// TwinCAT 3 PLC project CrimperProject
// ProgramVersion: 3.1.4023.0
// CompilerDefines: VISU_USEWSTRING, CRIMP_IO_TEST
// libraries:
//   CmpBitmapPool, * (System)
//   Tc2_Standard, * (Beckhoff Automation GmbH)
//   Tc2_System, * (Beckhoff Automation GmbH)
//   Tc2_Utilities, * (Beckhoff Automation GmbH)
//   Tc3_Module, * (Beckhoff Automation GmbH)
//   VisuDialogs, * (System)
//   VisuSymbols,3.5.10.0,System
// project tree:
//   DUTs/ DUT_Errors.TcDUT, DUT_Device.TcDUT, DUT_RunTime.TcDUT
//   / GlobalTextList.TcGTLO, ImagePool.TcIPO (not stored), PlcTask.TcTTO, VISU_TASK.TcTTO
//   GVLs/ CVL.TcGVL, DB6.TcGVL, GVL.TcGVL, IO.TcGVL, RVL.TcGVL, VAT.TcGVL
//   POUs/Helper/ FB_CalcXY.TcPOU, FB_INPUT_HANDLER.TcPOU, FB_MY_BLINK.TcPOU, P_GetTime.TcPOU, TSV.TcPOU
//   POUs/HMI/ P_HmiHandling.TcPOU
//   POUs/Initialization/ P_InitOnce.TcPOU
//   POUs/Language/ P_RestoreCurrentLanguage.TcPOU, P_SaveCurrentLanguage.TcPOU
//   POUs/ MAIN.TcPOU
//   POUs/MainPous/F20_Ablauf/AusstossVerzoegerung/ P_DecAusStossV.TcPOU, P_IncAusstossV.TcPOU
//   POUs/MainPous/F20_Ablauf/DrahtHalterDruck/ P_DecDruck.TcPOU, P_IncDruck.TcPOU
//   POUs/MainPous/F20_Ablauf/ F_AblaufketteLeerfahren.TcPOU, FB_AblaufketteNormal.TcPOU, P_AblaufReset.TcPOU, FB_AllesInSollposition.TcPOU, F_Endstellung.TcPOU, F_Ventile.TcPOU, P_Ablauf.TcPOU
//   POUs/MainPous/F20_Ablauf/SollwertRuettelTopf/ P_DecSollRuettel.TcPOU, P_IncSollRuettel.TcPOU
//   POUs/MainPous/FC24_Sortierer/ F_Leerfahren.TcPOU, F_Sortierer.TcPOU, F_Vereinzelung.TcPOU, P_Sortierer.TcPOU
//   POUs/MainPous/FC2_Betriebsarten/ P_BlinktaktTastleuchten.TcPOU, F_EndschalterBruecken.TcPOU, P_FlankenErzeugen.TcPOU, F_StartStopTipp.TcPOU, P_Betriebsarten.TcPOU, P_InputHandling.TcPOU, P_OutputHandling.TcPOU
//   POUs/MainPous/FC3_FehlerAllg/ F_Aufstarten.TcPOU, F_AusloeseschalterDauermeldung.TcPOU, F_Doppelmeldung.TcPOU, F_FehlerAufgetreten.TcPOU, F_GetErrorsAsDWORD.TcPOU, FB_KontrolleEndschalter.TcPOU, F_KontrollZeiten.TcPOU, F_ResetEndSchalterFehler.TcPOU, F_ResetErrors.TcPOU, F_StoerungsbitsAuswerten.TcPOU, P_FehlerAllgemein.TcPOU
//   POUs/MainPous/FC4_TpKommunikation/ F_AnzeigeNiedriegePrio.TcPOU, F_AnzeigeSollpositionsFehler.TcPOU, F_AuswertungBefehlstastenVonTP.TcPOU, F_SAFETY_AnzeigenHohePrio.TcPOU, F_SAFETY_AnzeigenHohePrio_Neu.TcPOU, F_SignaldauerVonTastleuchte_MaschEinAuswerten.TcPOU, P_OnResetClick.TcPOU, P_TpKommunikation.TcPOU
//   POUs/MainPous/FC95_StatusAnzeige/ P_StatusAnzeige.TcPOU
//   POUs/MainPous/FC99_LetzterFC/ P_LetzterFC.TcPOU
//   VISUs/ Ausstossverz.TcVIS, BetrAnzeigeListe.TcTLO, DrahthalterDruck.TcVIS, IO_Visu01.TcVIS, IO_Visu02.TcVIS, Menu.TcVIS, Probelauf.TcVIS, Rezeptur.TcVIS, Sprache.TcVIS, OutTest.TcVIS, SensorBruecken.TcVIS, Start.TcVIS, Stueckzahl.TcVIS, Total.TcVIS, VisualizationManager.TcVMO (not stored)
// real-time tasks:
//   TASK PlcTask: cycle T#20ms, priority 20, ADS port 350
//   TASK VISU_TASK: cycle T#200000us, priority 30, ADS port 351
//   TASK Standard: cycle T#1ms, priority 1, ADS port 352
//   TASK ELM-Task: cycle T#1ms, priority 2, ADS port 353
// I/O:
//   DEVICE Gerät 3 (EtherCAT), AmsNetId 172.18.216.102.4.1
//     Klemme 1 (EK1100-0008) [EK1100-0008 EtherCAT-Koppler M8 (2A E-Bus)]
//       Klemme 2 (EL1809) [EL1809 16K. Dig. Eingang 24V, 3ms]
//       Klemme 3 (EL2809) [EL2809 16K. Dig. Ausgang 24V, 0.5A]
//       Klemme 4 (EL4122) [EL4122 2K. Ana. Ausgang 4-20mA, 16bit]
//       Klemme 5 (EL2911) [EL2911,  Potential supply terminal (10 A) with 4 Ch. Safety Inputs, TwinSAFE]
//         modules: Module 2 (FSOUT), Module 3 (DEVICEIO), Module 4 (FSLOGIC)
//       Klemme 7 (ELM3702-0000) [ELM3702-0000 2K. Ana. Eingang +/-60V, +/-20mA, TC, RTD, Messbrückenauswertung (DMS), IEPE, 24 bit, hochgenau]
//       Klemme 6 (EL9011) [EL9011 Endklemme]
// variable links:
//   CrimperProject/CrimperProject Instance <-> Device 3 (EtherCAT)/Term 1 (EK1100-0008)/Term 2 (EL1809)
//     PlcTask Inputs/IO.inAbisoliererIstLINKS <-> Channel 8/Input
//     PlcTask Inputs/IO.inAbisoliererIstRUECK <-> Channel 7/Input
//     PlcTask Inputs/IO.inAbisoliererIstVORN <-> Channel 6/Input
//     PlcTask Inputs/IO.inAbisoliererIstZU <-> Channel 5/Input
//     PlcTask Inputs/IO.inAusloeseSchalter <-> Channel 4/Input
//     PlcTask Inputs/IO.inAusstossenVORN <-> Channel 14/Input
//     PlcTask Inputs/IO.inCrimpEinheitIstRUECK <-> Channel 13/Input
//     PlcTask Inputs/IO.inCrimpEinheitIstVORN <-> Channel 12/Input
//     PlcTask Inputs/IO.inCrimpZangeIstOFFEN <-> Channel 10/Input
//     PlcTask Inputs/IO.inCrimpZangeIstZU <-> Channel 9/Input
//     PlcTask Inputs/IO.inDrahthalterIstOffen <-> Channel 3/Input
//     PlcTask Inputs/IO.inKontaktIstGefallen <-> Channel 11/Input
//     PlcTask Inputs/IO.inKontaktSchiebenVORN <-> Channel 15/Input
//     PlcTask Inputs/IO.inMagazinGEFUELLT <-> Channel 16/Input
//     PlcTask Inputs/IO.inResetNotHalt <-> Channel 1/Input
//     PlcTask Inputs/IO.inStart <-> Channel 2/Input
//     PlcTask Inputs/IO.inWord0 @bit {1..15} <-> Channel {2..16}/Input  (15 links)
//     PlcTask Inputs/IO.inWord0 <-> Channel 1/Input
//   CrimperProject/CrimperProject Instance <-> Device 3 (EtherCAT)/Term 1 (EK1100-0008)/Term 3 (EL2809)
//     PlcTask Outputs/IO.outMldTasteStart <-> Channel 2/Output
//     PlcTask Outputs/IO.outNotHaltReset <-> Channel 1/Output
//     PlcTask Outputs/IO.outResA1_2 <-> Channel 3/Output
//     PlcTask Outputs/IO.outY10DrahthaltFuehrungZU <-> Channel 16/Output
//     PlcTask Outputs/IO.outY11SortierLuft <-> Channel 6/Output
//     PlcTask Outputs/IO.outY1Ausstossen <-> Channel 7/Output
//     PlcTask Outputs/IO.outY2KontaktVereinzelung <-> Channel 8/Output
//     PlcTask Outputs/IO.outY3KontaktSchieben <-> Channel 9/Output
//     PlcTask Outputs/IO.outY4CrimpEinheitVOR <-> Channel 10/Output
//     PlcTask Outputs/IO.outY5AbisolierNachLINKS <-> Channel 11/Output
//     PlcTask Outputs/IO.outY6AbisoliererZU <-> Channel 12/Output
//     PlcTask Outputs/IO.outY7AbfallRUNTER <-> Channel 13/Output
//     PlcTask Outputs/IO.outY8AbisoliererRUECK <-> Channel 14/Output
//     PlcTask Outputs/IO.outY9CrimperZU <-> Channel 15/Output
//   CrimperProject/CrimperProject Instance <-> Device 3 (EtherCAT)/Term 1 (EK1100-0008)/Term 4 (EL4122)
//     PlcTask Outputs/IO.outSollwertDruckVentil <-> Channel 2/Output
//     PlcTask Outputs/IO.outSollwertRuettelTopf <-> Channel 1/Output
//   CrimperProject/CrimperProject Instance <-> Device 3 (EtherCAT)/Term 1 (EK1100-0008)/Term 5 (EL2911)
//     PlcTask Inputs/IO.safeOutHauptLuft <-> StandardInputs/Standard Out Var 6
//     PlcTask Inputs/IO.safeOutNotHalt <-> StandardInputs/Standard Out Var 11
//     PlcTask Inputs/IO.safeOutSchutzTueren <-> StandardInputs/Standard Out Var 12
//     PlcTask Outputs/IO.safetyRUN <-> StandardOutputs/Standard In Var 2

CONFIGURATION CrimperProject
    RESOURCE PLC ON TwinCAT3
        TASK PlcTask(INTERVAL := T#20ms, PRIORITY := 20);
        TASK VISU_TASK(INTERVAL := T#200000us, PRIORITY := 30);
        PROGRAM MAIN WITH PlcTask : MAIN;
        PROGRAM VisuElems_Visu_Prg WITH VISU_TASK : VisuElems.Visu_Prg;
    END_RESOURCE
END_CONFIGURATION

// ---- DUTs/DUT_Errors.TcDUT
TYPE DUT_Errors :
STRUCT

    //M104.0
	DrahthltNichtOffen : BIT; //(ehem. M104.0) Drahthalter nicht offen, BetrAnzeigeListe.ID 600
	DrahthltNichtZu : BIT; //(ehem. M104.1) Drahthalter nicht zu, BetrAnzeigeListe.ID 601
	AusloesSchaltDauerMldg: BIT;//(ehem. M104.2) -- Auslöseschalter Dauermelung, BetrAnzeigeListe.ID 602
	AbisolierNichtOffen : BIT; //(ehem. M104.3) Abisolierer nicht offen, BetrAnzeigeListe.ID 603
	AbisolierNichtZu : BIT; //(ehem. M104.4) Abisolierer nicht zu, BetrAnzeigeListe.ID 604
	DoppelMlgAbisoVornRueck : BIT; //(ehem. M104.5) Doppelmeldung Abisolierer vorn+rück, BetrAnzeigeListe.ID 605
	AbisolierNichtVorn : BIT; //(ehem. M104.6) Abisolierer nicht vorn, BetrAnzeigeListe.ID 606
	AbisolierNichtRueck : BIT; //(ehem. M104.7) Abisolierer nicht rück (abisoliert), BetrAnzeigeListe.ID 607
	
	//M105.0
	AbisolierNichtLinks : BIT; //(ehem. M105.0) Abisolierer nicht links (aus Arbeitsraum) , BetrAnzeigeListe.ID 608
	AbisolierNichtRechts : BIT; //(ehem. M105.1) Abisolierer nicht rechts, BetrAnzeigeListe.ID 609
	DoppelMlgCrimpzZuOffen : BIT; //(ehem. M105.2) Doppelmeldung Crimpzange zu+offen, BetrAnzeigeListe.ID 610
	CrimpZangeNichtZu : BIT; //(ehem. M105.3) Crimpzange nicht zu, BetrAnzeigeListe.ID 611
	CrimpZangeNichtOffen : BIT; //(ehem. M105.4) Crimpzange nicht offen, BetrAnzeigeListe.ID 612
	KontaktNichtGefallen : BIT; //(ehem. M105.5) !! nur xls File !!, BetrAnzeigeListe.ID 613
	DauerMlgKontaktGefallen : BIT; //(ehem. 105.6) !! nur xls File !!, BetrAnzeigeListe.ID 614
	DoppelMlgCrimpEinhVornZurueck : BIT; //(ehem. M105.7) Doppelmeldung Crimpeinheit vorn+rück, BetrAnzeigeListe.ID 615
	
	//M106.0
	CrimpeinheitNichtVorn : BIT; //(ehem. M106.0)Crimpeinheit nicht vorn, BetrAnzeigeListe.ID 616
	CrimpeinheitNichtRueck : BIT; //(ehem. M106.1) Crimpeinheit nicht rück, BetrAnzeigeListe.ID 617
	KontaktSchiebenNichtVorn : BIT; //(ehem. M106.2) Kontakt-Schieben nicht vorn, BetrAnzeigeListe.ID 618
	KontaktSchiebenNichtRueck : BIT; //(ehem. M106.3) Kontakt-Schieben nicht rück, BetrAnzeigeListe.ID 619
	AusstossenNichtVorn : BIT; //(ehem. M106.4) Ausstoßen nicht vorn, BetrAnzeigeListe.ID 620
	AusstossenNichtRueck : BIT; //(ehem. M106.5) Ausstoßen nicht rück, BetrAnzeigeListe.ID 621
	r106_6 : BIT; //Reserve, war in AWL nicht belegt, BetrAnzeigeListe.ID 622
	WartungsZaehlErreicht : BIT; //(ehem. M106.7) Wartungs-Zähler, hat Vorwahl eicht, BetrAnzeigeListe.ID 623
	
	//M107.0
	StueckZaehlErreicht : BIT; //(ehem. M107.0 Stückzahl-Vorwahl eicht), BetrAnzeigeListe.ID 624
	r107_1 : BIT; //Reserve, war in AWL nicht belegt, BetrAnzeigeListe.ID 625 
	r107_2 : BIT; //Reserve, war in AWL nicht belegt, BetrAnzeigeListe.ID 626
	r107_3 : BIT; //Reserve, war in AWL nicht belegt, BetrAnzeigeListe.ID 627
	r107_4 : BIT; //Reserve, war in AWL nicht belegt, BetrAnzeigeListe.ID 628
	r107_5 : BIT; //Reserve, war in AWL nicht belegt, BetrAnzeigeListe.ID 629
	r107_6 : BIT; //Reserve, war in AWL nicht belegt, BetrAnzeigeListe.ID 630
	r107_7 : BIT; //Reserve, war in AWL nicht belegt, BetrAnzeigeListe.ID 631   

END_STRUCT
END_TYPE

// ---- DUTs/DUT_Device.TcDUT
TYPE DUT_Device :
STRUCT
	wID:WORD; (* Geräte ID *)
		
	rIN_LO:REAL; (* REAL in Wert unten *)
	rIN_HI:REAL; (* REAL in Wert oben *)
	nOUT_LO:UINT; (* RAW out Wert unten *)
	nOUT_HI:UINT; (* RAW out Wert oben *)
	
	dFakt_A:REAL; (* Faktor 'a' in Y=aX + b *)
	dSmd_B:REAL; (* Summand 'b' in Y=aX + b *)
	
	sDevName:STRING(50); (* Gerätename *)

END_STRUCT
END_TYPE

// ---- DUTs/DUT_RunTime.TcDUT
TYPE DUT_RunTime :
STRUCT
	seconds:INT;
	mins:INT;
	hours:DINT;
END_STRUCT
END_TYPE

// ---- GVLs/CVL.TcGVL
{attribute 'qualified_only'}
VAR_GLOBAL CONSTANT

(* LogLevels: 0-Nothing, 1-ErrOnly, 2-Warnings, 4-Info , 8-All *)
ERROR:WORD:=1;
WARNING:WORD:=2;
INFO:WORD:=4;
TRACE:WORD:=8;
	
enableIN1_2 : BOOL := TRUE; // (ehem. M11.0, insecDrahthalterIstOffen)

BTN_STOP : INT := 130; // Stop-Taste im Start-Menü ??? original ??? noch klären

BTRART_RESET : INT := 800; // Bertriebsarten-Reset 
RESET_BUTTON : INT := 801; // Reset-Button
MAGAZIN_LEER : INT := 810; // Magazin Leerfahren
SORTIER_LEER : INT := 820; // Sortierer Leerfahren
CRIMP_EINRICHTEN : INT := 830; //Crimpen Einrichten
NUR_ABISOLIER : INT := 840; // Nur Abisolieren
PROBE_OHNE_KONT : INT := 850; // Probelauf ohne Kontakt
PROBE_OHNE_CRIMP : INT := 860; // Probelauf ohne Crimpen
PROBE_OHNE_LITZE : INT :=870; // Probelauf ohne Litze
END_VAR

// ---- GVLs/DB6.TcGVL
{attribute 'qualified_only'}
VAR_GLOBAL RETAIN
	
	rAusstossverz : REAL := 0.0; //ehem. in DB6.w134
	nAusstossverz : INT := 0; //NEU-NBT

	diStueck_Vorwahl: DINT := 10000;//ehem. in DB6.d64Stueck_Vorwahl
	diStueck_Fertig: DINT := 0; //ehem. in DB6.d68Stueck_Fertig
	diStueck_Noch: DINT := 10000;
	iStueck_pro_Minute: INT := 0;
	
	diStueck_Total : DINT := 0;
	
	
	diTotalZaehler: DINT := 0; // ehem. in DB6.d140
	diTagesZaehler: DINT := 0; // ehem. in DB6.d144
	
	diWartZaehlVorwahl: DINT := 0; // Vorwahl Wartung, ehem. in DB6.d148
	diWartungsZaehler: DINT := 0; // ehem. in DB6.d152
	
	diReinigung_Vorw: DINT := 10000; //ehem. in DB6.d80
	diReinigung_Zaehl: DINT := 0; //ehem. in DB6.d84
	
	rDrahthalterSchliessdruck : REAL := 0.5; //Umwandlung in F_Ventile() - wDrahthalterSchliessdruck := REAL_TO_WORD(DINT_TO_REAL(DB6.d376) * 2.730000E+003);
	
	
	iSortierer : INT := 50; // Sortierer-Sollwert (Analog), war w132_Sortierer
	
	w226_Betr_Anz_Wert : INT := 0; // Betriebs-Anzeige-Wert Bedeutung noch unklar!!!
	w230 : INT := 0; // Signaldauer-Wert von PNOZ Bedeutung noch unklar!!!
	w228_Bef_Tast_Wert : INT := 0;
	
	outWordAlt : WORD; //ehem. in DB6.d408 -- Zuw.v. AW0
	
	d0 : DWORD := 0;
	
	runTime : DUT_RunTime;  //ehem. in DB6.d160 ff., todo versteckt. Reset?
	
	
	//Test später raus --- Begin ---
	
	frceY11SortierLuft 			: BOOL; //EL1809-A1.5
	frceY1Ausstossen 			: BOOL;
	frceY2KontaktVereinzelung 	: BOOL; //EL1809-A1.7
	frceY3KontaktSchieben	 	: BOOL; //EL1809-A1.8
	frceY4CrimpEinheitVOR	 	: BOOL; //EL1809-A1.9
	frceY5AbisolierNachLINKS	: BOOL; //EL1809-A1.10
	frceY6AbisoliererZU		 	: BOOL; //EL1809-A1.11
	frceY7AbfallRUNTER		 	: BOOL; //EL1809-A1.12
	frceY8AbisoliererRUECK	 	: BOOL; //EL1809-A1.13
	frceY9CrimperZU			 	: BOOL; //EL1809-A1.14
	frceY10DrahthaltFuehrungZU	: BOOL; //EL1809-A1.15
	
	//Test später raus --- End ---
END_VAR

// ---- GVLs/GVL.TcGVL
{attribute 'qualified_only'}
VAR_GLOBAL
	firstCycle : BOOL;	
	
	insecResetNotHalt			: BOOL; //result of P_InputHandling.E1_0
	insecTasterStart 			: BOOL; //result of P_InputHandling.E1_1
	insecDrahthalterIstOffen 	: BOOL; //result of P_InputHandling.E1_2
	insecAusloeseSchalter		: BOOL; //result of P_InputHandling.E1_3
	insecAbisoliererIstZU		: BOOL; //result of P_InputHandling.E1_4
	insecAbisoliererIstVORN		: BOOL; //result of P_InputHandling.E1_5
	insecAbisoliererIstRUECK	: BOOL; //result of P_InputHandling.E1_6
	insecAbisoliererIstLINKS	: BOOL; //result of P_InputHandling.E1_7
	
	insecCrimpZangeIstZU		: BOOL; //result of P_InputHandling.E1_8
	insecCrimpZangeIstOFFEN		: BOOL; //result of P_InputHandling.E1_9
	insecKontaktIstGefallen		: BOOL; //result of P_InputHandling.E1_10
	insecCrimpEinheitIstVORN	: BOOL; //result of P_InputHandling.E1_11
	insecCrimpEinheitIstRUECK	: BOOL; //result of P_InputHandling.E1_12
	insecAusstossenVORN			: BOOL; //result of P_InputHandling.E1_13
	insecKontaktSchiebenVORN	: BOOL; //result of P_InputHandling.E1_14
	insecMagazinGEFUELLT		: BOOL; //result of P_InputHandling.E1_15
	
	
	inTmpResetNotHalt			: BOOL; //result of P_InputHandling.E1_0
	inTmpTasterStart 			: BOOL; //result of P_InputHandling.E1_1
	inTmpDrahthalterIstOffen 	: BOOL; //result of P_InputHandling.E1_2
	inTmpAusloeseSchalter		: BOOL; //result of P_InputHandling.E1_3
	inTmpAbisoliererIstZU		: BOOL; //result of P_InputHandling.E1_4
	inTmpAbisoliererIstVORN		: BOOL; //result of P_InputHandling.E1_5
	inTmpAbisoliererIstRUECK	: BOOL; //result of P_InputHandling.E1_6
	inTmpAbisoliererIstLINKS	: BOOL; //result of P_InputHandling.E1_7
	
	inTmpCrimpZangeIstZU		: BOOL; //result of P_InputHandling.E1_8
	inTmpCrimpZangeIstOFFEN		: BOOL; //result of P_InputHandling.E1_9
	inTmpKontaktIstGefallen		: BOOL; //result of P_InputHandling.E1_10
	inTmpCrimpEinheitIstVORN	: BOOL; //result of P_InputHandling.E1_11
	inTmpCrimpEinheitIstRUECK	: BOOL; //result of P_InputHandling.E1_12
	inTmpAusstossenVORN			: BOOL; //result of P_InputHandling.E1_13
	inTmpKontaktSchiebenVORN	: BOOL; //result of P_InputHandling.E1_14
	inTmpMagazinGEFUELLT		: BOOL; //result of P_InputHandling.E1_15
	
	
	
	tof00Test : TOF;
	(* ehem. T0 ersetzt durch BLINK *)
	tonTasteStartOnErr : TON;	// (ehem. T1 SE->TON) Verzögerung Taste Start
	//T2 Verz.v. Taste Stop, existierte im AWL-Text nicht
	tonFehlerKontrMaschine  : TON; // (ehem. T3) Fehler-Kontr.Maschine (keine Bewegung)
	
	tonTasteStart : TON; // (ehem. T11) Taster-Start Verz. in F_Aufstarten(), für StörMldgLöschen
	tonBetrAnzeigReset : TON; // (ehem. T14) Verz. Betriebs-Anzeigen-Reset
	tonEndschalterBrueck : TON; // (ehem. T15) Verz. Endschalter-Brückung
	tonAusloesDauermld : TON; // (ehem. T16) Kontr.Auslöseschalter Dauermeldung
	tsvVereinzelZeit : TSV; // (ehem. T17) AWL-SV: Vereinzelungs-Zeit, Zeit mit verlängertem Impuls
	tonKontaktIstGefallen : TON; // (ehem. T18) Verz.v. E1.10 Kontakt gefallen
	tsvKontauswurf : TSV;	// (ehem. T19) AWL-SV: Kontaktauswurf nach Einschalten, Zeit mit verlängertem Impuls
	
	tofAblVerzProbelauf : TOF; 	// (ehem. T20) Ablauf-Verz.bei Probelauf
	ton2terVersuch : TON; //(ehem. T21) Verz. 2ter Vereinzelungs-Versuch
	tonAusstoss : TON; // (ehem. T22) Ausstoß-Verzögerung
	tonKontaktIstZuLangeEin : TON; //NEU Fehlererzeugung für DauermeldungKontaktGefallen
	
	tofCrimpzangeOffen : TOF; // (ehem. T31) Verl. E1.9 Crimpzange offen
	tofMagazGefuellt : TOF; // (ehem. T32) Verl. E1.15 Magazin gefüllt
	tofMagazGefuellt2 : TON; // (ehem. T33) 2te Verl. T32 E1.15 Magazin gefüllt
	
	tofBetrStdZaehl : TOF; // (ehem. T34)  Verl. 5 Minuten für Betriebstunden-Zähler, Zeit mit Ausschaltverzögerung
	tofMagazLeerFahr : TOF; // // (ehem. T41) Takt für Magazin leerfahren, wird 2x verwendet???

	
	tonResetNotHalt : TON; // Neu: check rote Stop-Taste
	//tonPnozEntprell  : TON; //(ehem. T70) PNOZ ???Entprell??
	//tofPnozSigLen : TOF; // (ehem. T71) PNOZ Signaldauer ???
	tonSAFETYok : TON; // (ehem. T72) Verzögerung Alles Ok von PNOZ, tonOkPNOZ
	
	
	tonDrahthaltOffen : TON; // (ehem. T110) Brücke EL1809-E1.2 Drahthalter offen
	tonAbisoliererIstZU : TON; // (ehem. T112) Brücke EL1809-E1.4 Abisolierer zu
	tonAbisoliererIstVORN : TON; // (ehem. T113) Brücke EL1809-E1.5 Abisolierer vorn
	tonAbisoliererIstRUECK : TON; // (ehem. T114) Brücke EL1809-E1.6 Abisolierer rück (abisoliert)
	tonAbisoliererIstLINKS : TON; // (ehem. T115) Brücke EL1809-E1.7 Abisolierer links (aus Arbeitsraum)
	tonCrimpZangeIstZU : TON; // (ehem. T116) Brücke EL1809-E1.8 Crimpzange zu
	tonCrimpZangeIstOFFEN : TON; // (ehem. T117) Brücke EL1809-E1.9 Crimpzange offen
	
	tonBrKontaktIstGefallen : TON; // (ehem. T120) Brücke EL1809-E1.10 Kontakt gefallen
	tonCrimpEinheitIstVORN : TON; // (ehem. T121) Brücke EL1809-E1.11 Crimpeinheit vorn
	tonKontaktSchiebenVORN : TON; // (ehem. T122) Brücke EL1809-E1.14 Kontakt-Schieben vorn
	tonAusstossenVORN : TON; // (ehem. T123) Brücke EL1809-E1.13 Ausstoßen vorn
	tonCrimpEinheitIstRUECK : TON; // (ehem. T124) Brücke EL1809-E1.12 Crimpeinheit rück
	
	bTEMP : BOOL;
	
	MW0 : WORD; //Bedeutung noch Unklar
	
	
	
	//MD20 : DWORD; //Bedeutung noch Unklar
	MD80 : DWORD; // +Fs ED0, wird offensichtlich nicht verwendet!	
		
	
	//MD100 : DWORD; //Bedeutung noch Unklar, irgendwas mit Störungen
	//MD104 : DWORD; //Bedeutung noch Unklar, irgendwas mit Störungen
	//MD108 : DWORD; //Bedeutung noch Unklar, irgendwas mit Störungen
	//MD112 : DWORD; //Bedeutung noch Unklar, irgendwas mit Störungen
	//MD116 : DWORD; //Bedeutung noch Unklar, irgendwas mit Störungen
	//MD120 : DWORD; //Bedeutung noch Unklar, irgendwas mit Störungen
	
	BetrAnzeigeIdx : INT; // (ehem. MW14 : WORD) // enthält Betriebs-Anzeige-Bits (jetzt Index)
	BetrAnzeigeTmp : INT;
	TopfWert : UINT;
	
	SolPosErrorIdx : WORD;
	EinzelschrittIdx : WORD;
	
	devSortierer : DUT_Device;
	devDruckVentil : DUT_Device;
	calcDev : FB_CalcXY;
	
	errs : DUT_Errors;
	errsAsDword : DWORD;
	zeigeFehler : BOOL;
	
END_VAR

// ---- GVLs/IO.TcGVL
{attribute 'qualified_only'}
VAR_GLOBAL

	//EL1809 16xDE (-10K1)
	inResetNotHalt				AT%I* : BOOL; //EL1809-E1.0 - roteTaste, LowAktiv
	inStart 					AT%I* : BOOL; //EL1809-E1.1 (ehem. E0.0)
	inDrahthalterIstOffen 		AT%I* : BOOL; //EL1809-E1.2 (ehem. E1.0)
	inAusloeseSchalter			AT%I* : BOOL; //EL1809-E1.3 (ehem. E1.1), wenn Draht in Aufnahme
	inAbisoliererIstZU			AT%I* : BOOL; //EL1809-E1.4 (ehem. E1.2)
	inAbisoliererIstVORN		AT%I* : BOOL; //EL1809-E1.5 (ehem. E1.3)
	inAbisoliererIstRUECK		AT%I* : BOOL; //EL1809-E1.6 (ehem. E1.4)
	inAbisoliererIstLINKS		AT%I* : BOOL; //EL1809-E1.7 (ehem. E1.5)
	
	inCrimpZangeIstZU			AT%I* : BOOL; //EL1809-E1.8 (ehem. E1.6)
	inCrimpZangeIstOFFEN		AT%I* : BOOL; //EL1809-E1.9 (ehem. E1.7)
	inKontaktIstGefallen		AT%I* : BOOL; //EL1809-E1.10 (ehem. E2.0)
	inCrimpEinheitIstVORN		AT%I* : BOOL; //EL1809-E1.11 (ehem. E2.1)
	inCrimpEinheitIstRUECK		AT%I* : BOOL; //EL1809-E1.12 (ehem. E2.4)
	inAusstossenVORN			AT%I* : BOOL; //EL1809-E1.13 (ehem. E2.3)
	inKontaktSchiebenVORN		AT%I* : BOOL; //EL1809-E1.14 (ehem. E2.2)
	inMagazinGEFUELLT			AT%I* : BOOL; //EL1809-E1.15 (ehem. E2.5)
	
	inWord0 					AT%I* : WORD; //Eingangswort komplett für EL1809-E1.
	
	
	
	//EL1809 16xDA (-10K4)
	outNotHaltReset 			AT%Q* : BOOL; //EL2809-A1.0
	//ToDo umben. 'TastleuchteStart'	
	outMldTasteStart			AT%Q* : BOOL; //EL2809-A1.1 (ehem. A0.0),Meldeleuchte Taste Start
	outResA1_2					AT%Q* : BOOL; //EL2809-A1.2
	//resA1.3
	//resA1.4
	outY11SortierLuft 			AT%Q* : BOOL; //EL2809-A1.5  (ehem. A0.1), toDo umben. BlasLuftSortierer...
	outY1Ausstossen 			AT%Q* : BOOL; //EL2809-A1.6  (ehem. A0.6)
	outY2KontaktVereinzelung	AT%Q* : BOOL; //EL2809-A1.7  (ehem. A0.7)
	outY3KontaktSchieben	 	AT%Q* : BOOL; //EL2809-A1.8  (ehem. A1.0)
	outY4CrimpEinheitVOR	 	AT%Q* : BOOL; //EL2809-A1.9  (ehem. A1.1)
	outY5AbisolierNachLINKS	 	AT%Q* : BOOL; //EL2809-A1.10 (ehem. A1.2)
	outY6AbisoliererZU		 	AT%Q* : BOOL; //EL2809-A1.11 (ehem. A1.3)
	outY7AbfallRUNTER		 	AT%Q* : BOOL; //EL2809-A1.12 (ehem. A1.4)
	outY8AbisoliererRUECK	 	AT%Q* : BOOL; //EL2809-A1.13 (ehem. A1.5)
	outY9CrimperZU			 	AT%Q* : BOOL; //EL2809-A1.14 (ehem. A1.6)
	outY10DrahthaltFuehrungZU	AT%Q* : BOOL; //EL2809-A1.15 (ehem. A1.7)
	
	
	//EL4122 (-10K6)
	outSollwertRuettelTopf		AT%Q* : UINT; //EL4122-AAW1
	//ToDo umbenennen bis in Klemme 4 outDrahthaltSchliessdrSoll
	outSollwertDruckVentil		AT%Q* : UINT; //EL4122-AAW2 Drahthalter Schliessdruck Sollwert
	
	//EL2911 (-10K6.1)
	safeInModuleFault			AT%I* : BOOL; //EL2911 In-Module-Fault
	safeOutNotHalt				AT%I* : BOOL; //EL2911 geklonter Ausgang des Not-Halt-AND Objekts
	safeOutSchutzTueren			AT%I* : BOOL; //EL2911 geklonter Ausgang des SchutzTueren-AND Objekts

	
	safeOutModuleFault			AT%I* : BOOL; //EL2911 Out-Module-Fault
	safeOutHauptLuft			AT%I* : BOOL; //EL2911-OUT1
	
	safetyErrAcknowledge 		AT%Q* : BOOL; //
	safetyRUN 					AT%Q* : BOOL; //EL2911 verlinkt mit dem Safety-Projekt 
	
	
	outWord0 : WORD; //Ausgangswort komplett für EL2809-E1. (selbst gefüllt)
END_VAR

// ---- GVLs/RVL.TcGVL
{attribute 'qualified_only'}
VAR_GLOBAL PERSISTENT
	
	e10Online : BOOL := TRUE; //ON-, OFF-line switch E1.0
	e11Online : BOOL := TRUE;
	e12Online : BOOL := TRUE;
	e13Online : BOOL := TRUE;
	e14Online : BOOL := TRUE;
	e15Online : BOOL := TRUE;
	e16Online : BOOL := TRUE;
	e17Online : BOOL := TRUE;
	
	e18Online : BOOL := TRUE;
	e19Online : BOOL := TRUE;
	e110Online : BOOL := TRUE; //ON-, OFF-line switch E1.10
	e111Online : BOOL := TRUE;
	e112Online : BOOL := TRUE;
	e113Online : BOOL := TRUE;
	e114Online : BOOL := TRUE;
	e115Online : BOOL := TRUE;
	
	e10OffMode : BOOL := FALSE; //Low-, High-switch for Offline mode E1.0
	e11OffMode : BOOL := FALSE;
	e12OffMode : BOOL := FALSE;
	e13OffMode : BOOL := FALSE;
	e14OffMode : BOOL := FALSE;
	e15OffMode : BOOL := FALSE;
	e16OffMode : BOOL := FALSE;
	e17OffMode : BOOL := FALSE;
		
	e18OffMode : BOOL := FALSE;
	e19OffMode : BOOL := FALSE;
	e110OffMode : BOOL := FALSE; //Low-, High-switch for Offline mode E1.10
	e111OffMode : BOOL := FALSE;
	e112OffMode : BOOL := FALSE;
	e113OffMode : BOOL := FALSE;
	e114OffMode : BOOL := FALSE;
	e115OffMode : BOOL := FALSE;

	
	currLogLevel : WORD := 0;
	currLanguage : STRING(10);
	
	
	//sBr: Sensor Brücke TRUE = eingeschalet, Sensor überbrückt
	sBrDrahthalterIstOffen 		: BOOL; //Brücke für: EL1809-E1.2
	sBrAusloeseSchalter			: BOOL; //Brücke für: EL1809-E1.3
	sBrAbisoliererIstZU			: BOOL; //Brücke für: EL1809-E1.4
	sBrAbisoliererIstVORN		: BOOL; //Brücke für: EL1809-E1.5
	sBrAbisoliererIstRUECK		: BOOL; //Brücke für: EL1809-E1.6
	sBrAbisoliererIstLINKS		: BOOL; //Brücke für: EL1809-E1.7
	
	sBrCrimpZangeIstZU			: BOOL; //Brücke für: EL1809-E1.8
	sBrCrimpZangeIstOFFEN		: BOOL; //Brücke für: EL1809-E1.9
	sBrKontaktIstGefallen		: BOOL; //Brücke für: EL1809-E1.10
	sBrCrimpEinheitIstVORN		: BOOL; //Brücke für: EL1809-E1.11
	sBrCrimpEinheitIstRUECK		: BOOL; //Brücke für: EL1809-E1.12
	sBrAusstossenVORN			: BOOL; //Brücke für: EL1809-E1.13
	sBrKontaktSchiebenVORN		: BOOL; //Brücke für: EL1809-E1.14
	sBrMagazinGEFUELLT			: BOOL; //Brücke für: EL1809-E1.15
END_VAR

// ---- GVLs/VAT.TcGVL
{attribute 'qualified_only'}
VAR_GLOBAL

	//MB5 : BYTE; // +F Blinktakt-Generator
	//MB6 : BYTE; // kein Gebrauch, nur 0-Initialisierung
	b00Test : BOOL := FALSE;
	//M0 : BYTE;
	(*
	0.0 -- frei
	0.1 -- frei
	0.2 -- 2te Ablauf-Freigabe
	0.3 -- Tipp, Einzel-Schritt
	0.4 -- frei 
	0.5 -- Bedingung für Ablauf-Freigabe
	0.6 -- SR Start
	0.7 -- Sammel-Störung
	*)
	bZweitAblaufFreig : BOOL; //ehem. M0.2 -- 2te Ablauf-Freigabe
 	bEinzelSchritt : BOOL;	//ehem. M0.3 -- Tipp, Einzel-Schritt
	bAblaufFreigabe : BOOL; //ehem. M0.5 -- Bedingung für Ablauf-Freigabe
	bSrStart : BOOL; 		//ehem. M0.6 -- SR Start
	bSammelStoerung : BOOL;	//ehem. M0.7 -- Sammel-Störung

	//M1 : BYTE;
	//1.0 -- frei 
	//1.1 -- frei
	//1.2 -- frei
	//1.3 -- RS Stop
	bRsStop : BOOL; //ehem. M1.3 -- RS Stop
	
	//M3 : BYTE;
	//3.0 -- Alles in Sollposition
	//3.1 -- PNOZ old
	//3.2 -- frei 
	//3.3 -- frei
	//3.4 -- frei
	//3.5 -- frei
	//3.6 -- frei
	//3.7 -- frei
	bAllesInSollPos : BOOL; //(ehem. M3.0 -- Alles in Sollposition)
	bResetNotHalt_Old : BOOL; //(ehem. M3.1 -- PNOZ old)
	
	//M4 : BYTE; //Blinktakt-Generator
	//4.0 -- 8-Hz Blinktakt
	//4.1 -- 4-Hz Blinktakt
	//4.2 -- 2-Hz Blinktakt
	//4.3 -- 1-Hz Blinktakt
	//4.4 -- 0.5-Hz Blinktakt (alle 2 sec)
	//4.5 -- 0.25-Hz Blinktakt (alle 4 sec)
	//4.6 -- 0.125-Hz Blinktakt (alle 8 sec)
	//4.7 -- frei
	
	byBlinkTakt : BYTE := 0; //Blinktakt-Generator (ehem. M4)
	//4.0 -- 8-Hz Blinktakt
	//4.1 -- 4-Hz Blinktakt
	//4.2 -- 2-Hz Blinktakt
	//4.3 -- 1-Hz Blinktakt
	//4.4 -- 0.5-Hz Blinktakt (alle 2 sec)
	//4.5 -- 0.25-Hz Blinktakt (alle 4 sec)
	//4.6 -- 0.125-Hz Blinktakt (alle 8 sec)
	//4.7 -- frei
		
	//M5 : BYTE;
	//5.0 
	//5.1
	//5.2
	//5.3 -- +F 1-Hz Blinktakt
	//5.4
	//5.5
	//5.6
	//5.7
	
	b1HzFlanke : BOOL; //(ehem. M5.3 -- +F 1-Hz Blinktakt)
	
	//M6 : BYTE;
	//6.0 -- +F Reset-Button
	bFlkResetButton : BOOL := FALSE; //(ehem. M6.0 -- +F Reset-Button)
	
	
	//M8 : BYTE; //MB8
	//8.0	M8.0 NormalCrimp
	//8.1	Magazin Leerfahren
	//8.2	Sortierer Leerfahren
	//8.3	"M8.3 CrimpEinr
	//8.4	"M8.4 NurAbisolieren
	//8.5	Probelauf ohne Kontakt
	//8.6	"M8.6 ohneCrmpen
	//8.7	"M8.7 Probelauf ohne Litze
	
	bNormalCrimp : BOOL; 			//(ehem. M8.0 NormalCrimp)
	bMagazinLeerfahren : BOOL; 		//(ehem. M8.1 Magazin Leerfahren)
	bSortiererLeerfahren : BOOL;	//(ehem. M8.2 Sortierer Leerfahren)
	bCrimpEinrichten : BOOL; 		//(ehem. M8.3 Crimp Einrichten)
	bNurAbisolieren : BOOL; 		//(ehem. M8.4 Nur Abisolieren)
	bProbelOhneKontakt : BOOL;		//(ehem. M8.5 Probelauf ohne Kontakt)
	bProbelOhneCrimpen : BOOL; 		//(ehem. M8.6 ohne Crimpen)
	bProbelOhneLitze : BOOL; 		//(ehem. M8.7 Probelauf ohne Litze)
	
	//M9 : BYTE;
	//9.0 -- mit Sortier-Blasen
	//9.1
	//9.2
	//9.3 
	//9.4
	//9.5
	//9.6
	//9.7
	bSortiererBlasen : BOOL; //(ehem. M9.0 -- mit Sortier-Blasen)
	bSortiererBlasenAlt : BOOL;
	sortierTextID : INT := 1000;
	
	//M11 : BYTE; --- RVL.sBrDrahthalterIstOffen...
	//11.0 -- Brücke E1.0 Drahthalter offen
	//11.1 -- Brücke E1.1 Auslöseschalter
	//11.2 -- Brücke E1.2 Abisolierer zu
	//11.3 -- Brücke E1.3 Abisolierer vorn
	//11.4 -- Brücke E1.4 Abisolierer rück (abisoliert)
	//11.5 -- Brücke E1.5 Abisolierer links (aus Arbeitsraum)
	//11.6 -- Brücke E1.6 Crimpzange zu
	//11.7 -- Brücke E1.7 Crimpzange offen
	
	// M12 : BYTE; --- RVL.sBrKontaktIstGefallen...
	//12.0 -- Brücke E2.0 Kontakt gefallen
	//12.1 -- Brücke E2.1 Crimpeinheit vorn
	//12.2 -- Brücke E2.2 Kontakt-Schieben vorn
	//12.3 -- Brücke E2.3 Ausstoßen vorn
	//12.4 -- Brücke E2.4 Crimpeinheit rück
	//12.5 -- Brücke E2.5 Magazin gefüllt
	//12.6
	//12.7
	
	//M14 : BYTE;
	//14.0 -- A55 Kontakt nicht gefallen
	//14.1
	//14.2
	//14.3
	//14.4
	//14.5
	//14.6
	//14.7
	bA55KontaktNichtGefallen:BOOL; //(ehem. M14.0 A55 Kontakt nicht gefallen)
	
	//M20 : BYTE; //Schrittkette
	//20.0 -- Drahthalter + Drahtführung zu
	//20.1 -- Abisolierer zu
	//20.2 -- Abisolierer rück
	//20.3 -- Abisolierer nach links + Abisolierer auf
	//20.4 -- Crimpeinheit vor
	//20.5 -- Crimpeinheit zu
	//20.6 -- Drahthalter + Drahtführung auf
	//20.7 -- Crimpzange auf + Abisoliereinheit vor
	
	bDrahtHalterUndFuehrungZU : BOOL; //(ehem. M20.0 -- Drahthalter + Drahtführung zu)
	bAbisoliererZU : BOOL; //(ehem. M20.1 -- Abisolierer zu )
	bAbisoliererRUECK : BOOL; //(ehem. M20.2 -- Abisolierer rück )
	bAbisoliererLINKSundAUF : BOOL; //(ehem. M20.3 -- Abisolierer nach links + Abisolierer auf )
	bCrimpeinheitVOR : BOOL; //(ehem. M20.4 --Crimpeinheit vor)
	bCrimpenZU : BOOL; //(ehem. M20.5 --Crimpeinheit zu)
	bDrahtHalterUndFuehrungAUF : BOOL; //(ehem. M20.6 --Drahthalter + Drahtführung auf)
	bCrZangeAUF_AisolierVOR : BOOL; //(ehem. M20.7 -- Crimpzange auf + Abisoliereinheit vor)
	
	
	//M21 : BYTE;
	//21.0  -- Ausstoßen vor
	//21.1 -- Crimpeinheit rück
	//21.2 -- Abisolierer nach rechts + Kontakt-Schieben rück
	//21.3
	//21.4
	//21.5
	//21.6 -- Aktueller Ablauf ohne Crimpen
	//21.7 -- Kontakt-Anforderung
	bAusstossenVOR : BOOL; //(ehem. M21.0 Ausstoßen vor)
	bCrimpeinheitRUECK : BOOL; //(ehem. M21.1 Ausstoßen vor)
	bAbisoNachRE_KontSchiebRUECK : BOOL; //(ehem. M21.2 Abisolierer nach rechts + Kontakt-Schieben rück)
	
	
	bAktAblaufOhneCr : BOOL;	//(ehem. M21.6  -- Aktueller Ablauf ohne Crimpen)
	bKontaktAnforderung : BOOL; //(ehem. M21.7  -- Kontakt-Anforderung)
	
	//M22 : BYTE;
	//22.0 -- Abisolierer nach Links Leerf-o-Crimpen
	//22.1 -- Crimpeinheit vor Leerf-o-Crimpen
	//22.2 -- Vereinzelung takten od.Crimpen
	//22.3 -- Crimpeinheit rück Leerf-o-Crimpen
	//22.4 -- frei
	//22.5 -- frei
	//22.6 -- Crimpen beim Einstellen
	//22.7 -- Endstellung
	bAbisoliererNachLinksLoC : BOOL; //(ehem. M22.0 Abisolierer nach Links Leerfahren-ohne-Crimpen)
	bCrimpEinheitVorLoC : BOOL; //(ehem. M22.1 Crimpeinheit vor Leerfahren-ohne-Crimpen)
	bVereinzelungTakten  : BOOL; //(ehem. M22.2 takten od.Crimpen)
	bCrimpEinheitRueckLoC : BOOL; //(ehem. M22.3 rück Leerfahren-ohne-Crimpen)
	//frei
	bCrimpenZuBeiEinstellen : BOOL; //(ehem. M22.6 Crimpen zu bei Einstellen Leerfahren-ohne-Crimpen)
	bEndstellung : BOOL; //(ehem. M22.7 Endstellung)
	
	//M23 : BYTE;
	//23.0 -- Takt für Vereinzelung bei Leerfahren
	//23.1 -- Zylinder sollen IN Leerfahrstellung
	//23.2 -- Zylinder sollen AUS Leerfahrstellung
	//23.3 -- S&R 2ter Vereinzelungs-Versuch
	//23.4
	//23.5
	//23.6
	//23.7
	bTaktVereinzLeerF : BOOL; //(ehem. M23.0 Takt für Vereinzelung bei Leerfahren)
	bZylINLeerFahrt : BOOL; //(ehem. M23.1 Zylinder sollen IN Leerfahrstellung)
	bZylAUSLeerFahrt : BOOL; //(ehem. M23.2 Zylinder sollen AUS Leerfahrstellung)
	bSr2terVereinzVersuch : BOOL; //(ehem. M23.3 S&R 2ter Vereinzelungs-Versuch)
	
	//M24 : BYTE;
	//24.0 
	//24.1 -- Zuw.v.T21 2ter Vereinzelungs-Versuch
	//24.2 -- +F 2ter Vereinzelungs-Versuch
	//24.3
	//24.4
	//24.5
	//24.6
	//24.7
	bFlk2terVersuch : BOOL; //(ehem. M24.2) +F 2ter Vereinzelungs-Versuch
	
	//M60 : BYTE; //MB60
	
	//M80 : BYTE;
	//80.0 //+F E0.0 Taste Start
	bFlkTasteStart : BOOL; //(ehem. M80.0) +F E0.0 Taste Start
	bFlkTasteStop : BOOL; //NEU
	
	//M81 : BYTE;
	//81.0 
	//81.1 -- +F E1.1 Auslöseschalter
	//81.2
	//81.3
	//81.4
	//81.5
	//81.6
	//81.7
	bFlankeAusloeseschalter : BOOL;  //(ehem. M81.1) +F E1.1 Auslöseschalter
	
	//M82 : BYTE;
	//82.0 
	//82.1 
	//82.2
	//82.3
	//82.4
	//82.5 -- +F E2.5 Magazin gefüllt
	//82.6
	//82.7
	bFlankeMagazGefuellt : BOOL; //(ehem. M82.5) +F E2.5 Magazin gefüllt
	
	(*
	
	//M104 : BYTE;
	//104.0 -- Drahthalter nicht offen
	//104.1 -- Drahthalter nicht zu
	//104.2 -- Auslöseschalter Dauermelung
	//104.3 -- Abisolierer nicht offen
	//104.4 -- Abisolierer nicht zu
	//104.5 -- Doppelmeldung Abisolierer vorn+rück
	//104.6 -- Abisolierer nicht vorn
	//104.7 -- Abisolierer nicht rück (abisoliert)
	errDrahthltNichtOffen : BOOL; //(ehem. M104.0) Drahthalter nicht offen
	errDrahthltNichtZu : BOOL; //(ehem. M104.1) Drahthalter nicht zu
	errAusloesSchaltDauerMldg: BOOL;//(ehem. M104.2) -- Auslöseschalter Dauermelung
	errAbisolierNichtOffen : BOOL; //(ehem. M104.3) Abisolierer nicht offen
	errAbisolierNichtZu : BOOL; //(ehem. M104.4) Abisolierer nicht zu
	errDoppelMlgAbisoVornRueck : BOOL; //(ehem. M104.5) Doppelmeldung Abisolierer vorn+rück
	errAbisolierNichtVorn : BOOL; //(ehem. M104.6) Abisolierer nicht vorn
	errAbisolierNichtRueck : BOOL; //(ehem. M104.7) Abisolierer nicht rück (abisoliert)
		
	
	//M105 : BYTE;
	//105.0 -- Abisolierer nicht links (aus Arbeitsraum)
	//105.1 -- Abisolierer nicht rechts
	//105.2 -- Doppelmeldung Crimpzange zu+offen
	//105.3 -- Crimpzange nicht zu
	//105.4 -- Crimpzange nicht offen
	//105.5 -- Kontakt nicht gefallen 
	//105.6
	//105.7 -- Doppelmeldung Crimpeinheit vorn+rück
	errAbisolierNichtLinks : BOOL; //(ehem. M105.0) Abisolierer nicht links (aus Arbeitsraum)
	errAbisolierNichtRechts : BOOL; //(ehem. M105.1) Abisolierer nicht rechts
	errDoppelMlgCrimpzZuOffen : BOOL; //(ehem. M105.2) Doppelmeldung Crimpzange zu+offen
	errCrimpZangeNichtZu : BOOL; //(ehem. M105.3) Crimpzange nicht zu
	errCrimpZangeNichtOffen : BOOL; //(ehem. M105.4) Crimpzange nicht offen
	errKontaktNichtGefallen : BOOL; //(ehem. M105.5) !! nur xls File !! --
	errDauermeldungKontaktGefallen : BOOL; //(ehem. 105.6) !! nur xls File !! --
	errDoppelMlgCrimpEinhVornZurueck : BOOL; //(ehem. M105.7) Doppelmeldung Crimpeinheit vorn+rück
	
	
	//M106 : BYTE;
	//106.0 -- Crimpeinheit nicht vorn
	//106.1 -- Crimpeinheit nicht rück
	//106.2 -- Kontakt-Schieben nicht vorn
	//106.3 -- Kontakt-Schieben nicht rück
	//106.4 -- Ausstoßen nicht vorn
	//106.5 -- Ausstoßen nicht rück
	//106.6
	//106.7 -- Wartungs-Zähler, hat Vorwahl erreicht, weiter mit Reset
	errCrimpeinheitNichtVorn : BOOL; //(ehem. M106.0)Crimpeinheit nicht vorn
	errCrimpeinheitNichtRueck : BOOL; //(ehem. M106.1) Crimpeinheit nicht rück
	errKontaktSchiebenNichtVorn : BOOL; //(ehem. M106.2) Kontakt-Schieben nicht vorn
	errKontaktSchiebenNichtRueck : BOOL; //(ehem. M106.3) Kontakt-Schieben nicht rück
	errAusstossenNichtVorn : BOOL; //(ehem. M106.4) Ausstoßen nicht vorn
	errAusstossenNichtRueck : BOOL; //(ehem. M106.5) Ausstoßen nicht rück
	//106.6
	bWartungsZaehlErreicht : BOOL := FALSE; //(ehem. M106.7) Wartungs-Zähler, hat Vorwahl erreicht
	
	//M107 : BYTE;
	//107.0 -- Stückzahl-Vorwahl erreicht
	//107.1 -- 
	//107.2 -- 
	//107.3 -- 
	//107.4 -- 
	//107.5
	//107.6
	//107.7
	bStueckZaehlErreicht : BOOL := FALSE; //(ehem. M107.0 Stückzahl-Vorwahl erreicht)
	*)
	aw4Sortierer : WORD;
END_VAR

// ---- POUs/MAIN.TcPOU
PROGRAM MAIN
VAR
	//rTrig : R_TRIG;
	dwTmp : DWORD;
END_VAR

P_InitOnce(); // NBT-NEU 

P_GetTime(); // NBT-NEU 

P_RestoreCurrentLanguage(); // NBT-NEU 

P_InputHandling(); // NBT-NEU 

P_TpKommunikation(); //ehem. FC4 -- OK

P_Betriebsarten(); //ehem. FC2 -- OK

P_Ablauf(); //ehem. FC20 -- OK -- 500er ID-Bereich

P_Sortierer(); //ehem. FC24 -- OK

P_FehlerAllgemein(); //ehem. FC3 -- OK -- 600er ID-Bereich

P_StatusAnzeige(); //ehem. FC95

//P_LetzterFC(); //ehem. FC99

P_OutputHandling(); // OK

P_HmiHandling(); //NBT-NEU

METHOD M_Log : DINT
VAR_INPUT
	reqLevel : WORD; (* 0-Nothing, 1-ErrOnly, 2-Warnings, 4-Info , 8-Verbose *)
	objectName : STRING(40);
	sMsg	: T_MaxString;(* Message string *)
	errNo : UDINT := 16#FFFFFFFF;
END_VAR
VAR
	sTmp : STRING;
END_VAR
IF WORD_TO_BOOL(RVL.currLogLevel AND reqLevel) = TRUE THEN
	
	sTmp := '[';
	sTmp := CONCAT( sTmp, objectName);
	sTmp := CONCAT( sTmp, '], ');
	
	CASE reqLevel OF
	 1:  sTmp := CONCAT( sTmp,'[E] ');
	 2:  sTmp := CONCAT( sTmp,'[W] ');
	 4:  sTmp := CONCAT( sTmp,'[I] ');
	 8:  sTmp := CONCAT( sTmp,'[T] ');
	ELSE 
		sTmp := CONCAT( sTmp,'[...] ');
	END_CASE 

	IF errNo <> 16#FFFFFFFF THEN
		sMsg := CONCAT( sMsg,': ');
		sMsg := CONCAT( sMsg, UDINT_TO_STRING(errNo));
	END_IF
	(*
	{IF defined (LOG_VIA_TCP)}
		LOG_PUSH_MSG(msg := CONCAT( sTmp, sMsg));
	{END_IF}
	*)
	M_Log := ADSLOGSTR( ADSLOG_MSGTYPE_HINT OR ADSLOG_MSGTYPE_LOG, CONCAT( sTmp, '%s' ), sMsg );
END_IF
END_METHOD

END_PROGRAM

// ---- POUs/Initialization/P_InitOnce.TcPOU
PROGRAM P_InitOnce
VAR
	done : BOOL;
	
END_VAR

GVL.firstCycle := FALSE;

IF done THEN
	RETURN;
END_IF

done := TRUE;

GVL.firstCycle := TRUE;


GVL.devSortierer.wID := 100;
GVL.devSortierer.sDevName := 'Sortierer';
GVL.devSortierer.rIN_LO := 0;
GVL.devSortierer.rIN_HI := 100; //ToDo: Checken
GVL.devSortierer.nOUT_LO := 819;
GVL.devSortierer.nOUT_HI := 65535;
GVL.calcDev(Dev := ADR(GVL.devSortierer));

GVL.devDruckVentil.wID := 101;
GVL.devDruckVentil.sDevName := 'Druck-Ventil';
GVL.devDruckVentil.rIN_LO := 0.0;
GVL.devDruckVentil.rIN_HI := 100.0;
GVL.devDruckVentil.nOUT_LO := 0;
GVL.devDruckVentil.nOUT_HI := 65535;
GVL.calcDev(Dev := ADR(GVL.devDruckVentil));


VAT.byBlinkTakt := 0;

DB6.runTime.seconds := 0;

//Später wieder raus
VAT.bSammelStoerung := 0;

RVL.currLogLevel := 8;

DB6.nAusstossverz := REAL_TO_INT(DB6.rAusstossverz * 1000);

MAIN.M_Log(reqLevel:=CVL.INFO, objectName:= 'P_InitOnce', sMsg:='done', errNo:= 0);

IO.safetyRUN := TRUE;

END_PROGRAM

// ---- POUs/Helper/P_GetTime.TcPOU
PROGRAM P_GetTime
VAR
	fbGetLocalTime  : NT_GetTime;
    bBusy           : BOOL;
    bError          : BOOL;
    nErrID          : UDINT;
    presetTime      : TIMESTRUCT;

    syncTimer       : TON;
    syncTrigger     : F_TRIG;
    bSynchronize    : BOOL;    
    
    fbRTC           : RTC;
    bValid_RTC      : BOOL;
    time_RTC        : DT;
END_VAR

syncTimer(IN:= NOT syncTimer.Q, PT:= T#500MS);

fbGetLocalTime(START:=syncTimer.Q,NETID:='',TMOUT:=T#500MS, TIMESTR => presetTime);

syncTrigger(CLK := fbGetLocalTime.BUSY AND NOT fbGetLocalTime.ERR, Q => bSynchronize);

fbRTC(EN := bSynchronize, PDT := SYSTEMTIME_TO_DT(TIMESTR:= presetTime), Q => bValid_RTC, CDT => time_RTC);

END_PROGRAM

// ---- POUs/Language/P_RestoreCurrentLanguage.TcPOU
PROGRAM P_RestoreCurrentLanguage
VAR
	waitTon:TON;
	langDone:bool := FALSE;
END_VAR

waitTon(IN:=NOT langDone, PT:=T#8S);

IF waitTon.Q AND NOT langDone THEN
	langDone := TRUE;
	
	//MAIN.M_Log(reqLevel:=CVL.INFO, objectName:= 'P_RestoreCurrentLanguage', sMsg:=RVL.currLanguage, errNo:= 0);
	
	IF RVL.currLanguage <> '' THEN
		VisuElems.CurrentLanguage := RVL.currLanguage;
	ELSE
		VisuElems.CurrentLanguage := 'de';
	END_IF
	
	MAIN.M_Log(reqLevel:=CVL.INFO, objectName:= 'P_RestoreCurrentLanguage', sMsg:= CONCAT('Language = ', RVL.currLanguage), errNo:= 0);
END_IF

END_PROGRAM

// ---- POUs/MainPous/FC2_Betriebsarten/P_InputHandling.TcPOU
PROGRAM P_InputHandling
VAR
	rTrigStart : R_TRIG;
	fTrigStop : F_TRIG;
	nTmp : INT := 0;
	
	
	(* E1_0 : FB_INPUT_HANDLER;
	E1_1 : FB_INPUT_HANDLER; *)
	E1_2 : FB_INPUT_HANDLER;
	E1_3 : FB_INPUT_HANDLER;
	E1_4 : FB_INPUT_HANDLER;
	E1_5 : FB_INPUT_HANDLER;
	E1_6 : FB_INPUT_HANDLER;
	E1_7 : FB_INPUT_HANDLER;

	E1_8 : FB_INPUT_HANDLER;
	E1_9 : FB_INPUT_HANDLER;
	E1_10 : FB_INPUT_HANDLER;
	E1_11 : FB_INPUT_HANDLER;
	E1_12 : FB_INPUT_HANDLER;
	E1_13 : FB_INPUT_HANDLER;
	E1_14 : FB_INPUT_HANDLER;
	E1_15 : FB_INPUT_HANDLER; 
	
	inWordOld : WORD;
	
	inTmpE1_2old : BOOL;
	inTmpE1_3old : BOOL;
	inTmpE1_4old : BOOL;
	inTmpE1_5old : BOOL;
	inTmpE1_6old : BOOL;
	inTmpE1_7old : BOOL;
	
	inTmpE1_8old : BOOL;
	inTmpE1_9old : BOOL;
	inTmpE1_10old : BOOL;
	inTmpE1_11old : BOOL;
	inTmpE1_12old : BOOL;
	inTmpE1_13old : BOOL;
	inTmpE1_14old : BOOL;
	inTmpE1_15old : BOOL;
	
END_VAR

GVL.insecTasterStart := IO.inStart;

GVL.tonSAFETYok(IN := IO.safeOutHauptLuft, PT := T#1S);

{IF defined (CRIMP_IO_TEST)}
(*
E1_0(orgIN := IO.inResetNotHalt, onlineSwitch := RVL.e10Online, offLineState := RVL.e10OffMode,
	resultIN => GVL.inTmpResetNotHalt); 
	
E1_1(orgIN := IO.inStart, onlineSwitch := RVL.e11Online, offLineState := RVL.e11OffMode,
	resultIN => GVL.inTmpTasterStart);
*)
E1_2(orgIN := IO.inDrahthalterIstOffen, onlineSwitch := RVL.e12Online, offLineState := RVL.e12OffMode,
	resultIN => GVL.inTmpDrahthalterIstOffen);

E1_3(orgIN := IO.inAusloeseSchalter, onlineSwitch := RVL.e13Online, offLineState := RVL.e13OffMode,
	resultIN => GVL.inTmpAusloeseSchalter);

E1_4(orgIN := IO.inAbisoliererIstZU, onlineSwitch := RVL.e14Online, offLineState := RVL.e14OffMode,
	resultIN => GVL.inTmpAbisoliererIstZU);

E1_5(orgIN := IO.inAbisoliererIstVORN, onlineSwitch := RVL.e15Online, offLineState := RVL.e15OffMode,
	resultIN => GVL.inTmpAbisoliererIstVORN);

E1_6(orgIN := IO.inAbisoliererIstRUECK, onlineSwitch := RVL.e16Online, offLineState := RVL.e16OffMode,
	resultIN => GVL.inTmpAbisoliererIstRUECK);

E1_7(orgIN := IO.inAbisoliererIstLINKS, onlineSwitch := RVL.e17Online, offLineState := RVL.e17OffMode,
	resultIN => GVL.inTmpAbisoliererIstLINKS);
	
//-------------	
	
E1_8(orgIN := IO.inCrimpZangeIstZU, onlineSwitch := RVL.e18Online, offLineState := RVL.e18OffMode,
	resultIN => GVL.inTmpCrimpZangeIstZU);
	
E1_9(orgIN := IO.inCrimpZangeIstOFFEN, onlineSwitch := RVL.e19Online, offLineState := RVL.e19OffMode,
	resultIN => GVL.inTmpCrimpZangeIstOFFEN);

E1_10(orgIN := IO.inKontaktIstGefallen, onlineSwitch := RVL.e110Online, offLineState := RVL.e110OffMode,
	resultIN => GVL.inTmpKontaktIstGefallen);

E1_11(orgIN := IO.inCrimpEinheitIstVORN, onlineSwitch := RVL.e111Online, offLineState := RVL.e111OffMode,
	resultIN => GVL.inTmpCrimpEinheitIstVORN);

E1_12(orgIN := IO.inCrimpEinheitIstRUECK, onlineSwitch := RVL.e112Online, offLineState := RVL.e112OffMode,
	resultIN => GVL.inTmpCrimpEinheitIstRUECK);

E1_13(orgIN := IO.inAusstossenVORN, onlineSwitch := RVL.e113Online, offLineState := RVL.e113OffMode,
	resultIN => GVL.inTmpAusstossenVORN);

E1_14(orgIN := IO.inKontaktSchiebenVORN, onlineSwitch := RVL.e114Online, offLineState := RVL.e114OffMode,
	resultIN => GVL.inTmpKontaktSchiebenVORN);

E1_15(orgIN := IO.inMagazinGEFUELLT, onlineSwitch := RVL.e115Online, offLineState := RVL.e115OffMode,
	resultIN => GVL.inTmpMagazinGEFUELLT);
{END_IF}

IF inWordOld <> IO.inWord0 THEN
	
	MAIN.M_Log(reqLevel:=CVL.TRACE, objectName:= 'IN', sMsg:= '--------',errNo := 16#FFFFFFFF);
	
	IF inTmpE1_2old <> GVL.inTmpDrahthalterIstOffen THEN
		MAIN.M_Log(reqLevel:=CVL.TRACE, objectName:= 'IN', sMsg:= 'DrahthalterIstOffen', errNo:= BOOL_TO_UDINT(GVL.inTmpDrahthalterIstOffen));
	END_IF
	inTmpE1_2old := GVL.inTmpDrahthalterIstOffen;
	
	IF inTmpE1_3old <> GVL.inTmpAusloeseSchalter THEN
		MAIN.M_Log(reqLevel:=CVL.TRACE, objectName:= 'IN', sMsg:= 'AusloeseSchalter', errNo:= BOOL_TO_UDINT(GVL.inTmpAusloeseSchalter));
	END_IF
	inTmpE1_3old := GVL.inTmpAusloeseSchalter;
	
	IF inTmpE1_4old <> GVL.inTmpAbisoliererIstZU THEN	
		MAIN.M_Log(reqLevel:=CVL.TRACE, objectName:= 'IN', sMsg:= 'AbisoliererIstZU', errNo:= BOOL_TO_UDINT(GVL.inTmpAbisoliererIstZU));
	END_IF
	inTmpE1_4old := GVL.inTmpAbisoliererIstZU;
	
	IF inTmpE1_5old <> GVL.inTmpAbisoliererIstVORN THEN	
		MAIN.M_Log(reqLevel:=CVL.TRACE, objectName:= 'IN', sMsg:= 'AbisoliererIstVORN', errNo:= BOOL_TO_UDINT(GVL.inTmpAbisoliererIstVORN));
	END_IF
	inTmpE1_5old := GVL.inTmpAbisoliererIstVORN;
	
	IF inTmpE1_6old <> GVL.inTmpAbisoliererIstRUECK THEN	
		MAIN.M_Log(reqLevel:=CVL.TRACE, objectName:= 'IN', sMsg:= 'AbisoliererIstRUECK', errNo:= BOOL_TO_UDINT(GVL.inTmpAbisoliererIstRUECK));
	END_IF
	inTmpE1_6old := GVL.inTmpAbisoliererIstRUECK;
	
	IF inTmpE1_7old <> GVL.inTmpAbisoliererIstLINKS THEN	
		MAIN.M_Log(reqLevel:=CVL.TRACE, objectName:= 'IN', sMsg:= 'AbisoliererIstLINKS', errNo:= BOOL_TO_UDINT(GVL.inTmpAbisoliererIstLINKS));
	END_IF
	inTmpE1_7old := GVL.inTmpAbisoliererIstLINKS;
		
	
	IF inTmpE1_8old <> GVL.inTmpCrimpZangeIstZU THEN	
		MAIN.M_Log(reqLevel:=CVL.TRACE, objectName:= 'IN', sMsg:= 'CrimpZangeIstZU', errNo:= BOOL_TO_UDINT(GVL.inTmpCrimpZangeIstZU));
	END_IF
	inTmpE1_8old := GVL.inTmpCrimpZangeIstZU;
	
	IF inTmpE1_9old <> GVL.inTmpCrimpZangeIstOFFEN THEN	
		MAIN.M_Log(reqLevel:=CVL.TRACE, objectName:= 'IN', sMsg:= 'CrimpZangeIstOFFEN', errNo:= BOOL_TO_UDINT(GVL.inTmpCrimpZangeIstOFFEN));
	END_IF
	inTmpE1_9old := GVL.inTmpCrimpZangeIstOFFEN;
	
	IF inTmpE1_10old <> GVL.inTmpKontaktIstGefallen THEN	
		MAIN.M_Log(reqLevel:=CVL.TRACE, objectName:= 'IN', sMsg:= 'KontaktIstGefallen', errNo:= BOOL_TO_UDINT(GVL.inTmpKontaktIstGefallen));
	END_IF
	inTmpE1_10old := GVL.inTmpKontaktIstGefallen;
	
	IF inTmpE1_11old <> GVL.inTmpCrimpEinheitIstVORN THEN	
		MAIN.M_Log(reqLevel:=CVL.TRACE, objectName:= 'IN', sMsg:= 'CrimpEinheitIstVORN', errNo:= BOOL_TO_UDINT(GVL.inTmpCrimpEinheitIstVORN));
	END_IF
	inTmpE1_11old := GVL.inTmpCrimpEinheitIstVORN;
	
	IF inTmpE1_12old <> GVL.inTmpCrimpEinheitIstRUECK THEN	
		MAIN.M_Log(reqLevel:=CVL.TRACE, objectName:= 'IN', sMsg:= 'CrimpEinheitIstRUECK', errNo:= BOOL_TO_UDINT(GVL.inTmpCrimpEinheitIstRUECK));
	END_IF
	inTmpE1_12old := GVL.inTmpCrimpEinheitIstRUECK;
	
	IF inTmpE1_13old <> GVL.inTmpAusstossenVORN THEN	
		MAIN.M_Log(reqLevel:=CVL.TRACE, objectName:= 'IN', sMsg:= 'AusstossenVORN', errNo:= BOOL_TO_UDINT(GVL.inTmpAusstossenVORN));
	END_IF
	inTmpE1_13old := GVL.inTmpAusstossenVORN;
	
	IF inTmpE1_14old <> GVL.inTmpAbisoliererIstLINKS THEN	
		MAIN.M_Log(reqLevel:=CVL.TRACE, objectName:= 'IN', sMsg:= 'KontaktSchiebenVORN', errNo:= BOOL_TO_UDINT(GVL.inTmpKontaktSchiebenVORN));
	END_IF
	inTmpE1_14old := GVL.inTmpAbisoliererIstLINKS;
	
	IF inTmpE1_15old <> GVL.inTmpMagazinGEFUELLT THEN	
		MAIN.M_Log(reqLevel:=CVL.TRACE, objectName:= 'IN', sMsg:= 'MagazinGEFUELLT', errNo:= BOOL_TO_UDINT(GVL.inTmpMagazinGEFUELLT));
	END_IF
	inTmpE1_15old := GVL.inTmpMagazinGEFUELLT;
END_IF

inWordOld := IO.inWord0;

//------- neu --- 2021-01-22
//diese Funktionalität war nicht zu finden. ToDo: check ob nicht GVL.inTmpTasterStart direkt verwendet werden soll

rTrigStart( CLK := GVL.insecTasterStart);
VAT.bFlkTasteStart := rTrigStart.Q;


fTrigStop(CLK := IO.inResetNotHalt);
VAT.bFlkTasteStop := fTrigStop.Q;
IF VAT.bFlkTasteStop THEN
	nTmp := nTmp + 1;
	 P_OnResetClick();
END_IF

//------- neu ---

END_PROGRAM

// ---- POUs/Helper/FB_INPUT_HANDLER.TcPOU
FUNCTION_BLOCK FB_INPUT_HANDLER
VAR_INPUT
	orgIN : BOOL;
	onlineSwitch : BOOL;
	offLineState : BOOL;
END_VAR
VAR_OUTPUT
	resultIN : BOOL;
	onlineImageID : STRING(20);
 	modeImageID : STRING(20);
END_VAR
VAR
	orgIN_old : BOOL;
	onlineSwitch_old : BOOL;
	offLineState_old : BOOL;
END_VAR

IF GVL.firstCycle THEN
	
	IF onlineSwitch THEN
		onlineImageID := 'switch_on';
		modeImageID := 'switch_undef';
	ELSE
		onlineImageID := 'switch_off';
		
		IF offLineState THEN
			modeImageID := 'switch_on';
		ELSE
			modeImageID := 'switch_off';
		END_IF
		
	END_IF
	
	
	
END_IF

IF onlineSwitch THEN
	resultIN := orgIN;
	IF onlineSwitch <> onlineSwitch_old THEN
		onlineImageID := 'switch_on';
		modeImageID := 'switch_undef';
	END_IF
	
	offLineState := FALSE;
	(* IF offLineState <> offLineState_old THEN
		modeImageID := 'switch_undef';
	END_IF *)
	
ELSE	
	IF onlineSwitch <> onlineSwitch_old THEN
		onlineImageID := 'switch_off';
	END_IF

	IF offLineState THEN
		resultIN := TRUE;
		IF offLineState <> offLineState_old THEN
			modeImageID := 'switch_on';
		END_IF
	ELSE
		resultIN := FALSE;
		IF offLineState <> offLineState_old THEN
			modeImageID := 'switch_off';
		END_IF
	END_IF

END_IF
orgIN_old := orgIN;
onlineSwitch_old := onlineSwitch;
offLineState_old := offLineState;

END_FUNCTION_BLOCK

// ---- POUs/MainPous/FC4_TpKommunikation/P_OnResetClick.TcPOU
PROGRAM P_OnResetClick
VAR
END_VAR

F_AuswertungBefehlstastenVonTP(tastenWert := CVL.RESET_BUTTON);
F_ResetEndSchalterFehler();

END_PROGRAM

// ---- POUs/MainPous/FC4_TpKommunikation/F_AuswertungBefehlstastenVonTP.TcPOU
FUNCTION F_AuswertungBefehlstastenVonTP : BOOL
VAR_INPUT
	tastenWert : INT;
END_VAR
VAR
END_VAR

(* Netzwerk: 1 ===============================================================================================
Auswertung Befehlstasten von TP *)


//L 0  -- Lade die Zahl in AKKU 1 und schiebe aktuelles in AKKU 2
//T "MB 6" MB6 --Bits zurück auf 0
//VAT.MB6 := 0; //Bits zurück auf 0 -- soweit KEINE VERWENDUNG zu erkennen

DB6.w228_Bef_Tast_Wert := tastenWert;
//L "DB6".w228_Bef_Tast_Wert DB6.DBW228 -- Befehlstasten-Wert
//L 0
//==I
//SPB Aend // Springe wenn VKE = 1 (VKE: Verknüpfungsergebnis) 

IF DB6.w228_Bef_Tast_Wert = 0 THEN
	RETURN;
END_IF


//L "DB6".w228_Bef_Tast_Wert DB6.DBW228 -- Befehlstasten-Wert
//L 30 //*** Tipp/Auto
//==I
//SPBN b30 // Springe wenn VKE = 0

//UN "M0_3_Tipp" M0.3 -- Einzel-Schritt // UND NICHT
//= "M0_3_Tipp" M0.3 -- Einzel-Schritt // Zuweisung, Bitverknüpfung

//...springe nicht -> wenn gleich
IF DB6.w228_Bef_Tast_Wert = 30 THEN //*** Tipp/Auto 
	VAT.bEinzelSchritt := NOT VAT.bEinzelSchritt; //Einzel-Schritt
END_IF

//b30: BLD 130 //Sprungadresse

//L "DB6".w228_Bef_Tast_Wert DB6.DBW228 -- Befehlstasten-Wert
//L 130 //*** Bertriebsarten-Reset
//==I
//SPBN b130 // Springe wenn VKE = 0
//S "M1.3_Stop" M1.3 -- RS Stop

//...springe nicht -> wenn gleich
IF DB6.w228_Bef_Tast_Wert = 130 THEN // *** Bertriebsarten-Reset
	VAT.bRsStop := TRUE;
END_IF


//b130: BLD 130  //Sprungadresse

//L "DB6".w228_Bef_Tast_Wert DB6.DBW228 -- Befehlstasten-Wert
//L 800 (*** Bertriebsarten-Reset *)
//==I
//SPBN b800
//R "M0.6" M0.6 -- SR Start
//S "M 6.0" M6.0 -- +F Reset-Button
//R "M8.1MagLeerf" M8.1 -- Magazin Leerfahren
//R "M8.2SortLeerf" M8.2 -- Sortierer Leerfahren
//R "M8.3CrimpEinr" M8.3 -- Crimpen Einrichten
//R "M8.4NurAbisolieren" M8.4 -- Nur Abisolieren
//R "M8.5ohneKontakt" M8.5 -- Probelauf ohne Kontakt
//R "M8.6ohneCrmpen" M8.6 -- Probelauf ohne Crimpen
//R "M8.7ohneLitze" M8.7 -- Probelauf ohne Litze

//...springe nicht -> wenn gleich
IF DB6.w228_Bef_Tast_Wert = 800 THEN  //*** Bertriebsarten-Reset 
	VAT.bSrStart := FALSE; //SR Start
	VAT.bFlkResetButton := TRUE; //+F Reset-Button
	
	VAT.bMagazinLeerfahren := FALSE; //Reset ...see above.
	VAT.bSortiererLeerfahren := FALSE;
	VAT.bCrimpEinrichten := FALSE;
	VAT.bNurAbisolieren := FALSE;
	VAT.bProbelOhneKontakt := FALSE;
	VAT.bProbelOhneCrimpen := FALSE;
	VAT.bProbelOhneLitze := FALSE;
END_IF

//b800: BLD 130 //Sprungadresse

//L "DB6".w228_Bef_Tast_Wert DB6.DBW228 -- Befehlstasten-Wert
//L 801 //*** Reset-Button
//==I
//SPBN b801
//R "M0.6" M0.6 -- SR Start
//S "M1.3_Stop" M1.3 -- RS Stop
//S "M 6.0" M6.0 -- +F Reset-Button
//R "M8.1MagLeerf" M8.1 -- Magazin Leerfahren
//R "M8.2SortLeerf" M8.2 -- Sortierer Leerfahren
//R "M8.3CrimpEinr" M8.3 -- Crimpen Einrichten
//R "M8.4NurAbisolieren" M8.4 -- Nur Abisolieren
//R "M8.5ohneKontakt" M8.5 -- Probelauf ohne Kontakt
//R "M8.6ohneCrmpen" M8.6 -- Probelauf ohne Crimpen
//R "M8.7ohneLitze" M8.7 -- Probelauf ohne Litze

//...springe nicht -> wenn gleich
IF DB6.w228_Bef_Tast_Wert = 801 THEN //*** Reset-Button
	VAT.bSrStart := FALSE; //SR Start
	VAT.bRsStop := TRUE; //RS Stop
	VAT.bFlkResetButton := TRUE; //+F Reset-Button
	
	VAT.bMagazinLeerfahren := FALSE;
	VAT.bSortiererLeerfahren := FALSE;
	VAT.bCrimpEinrichten := FALSE;
	VAT.bNurAbisolieren := FALSE;
	VAT.bProbelOhneKontakt := FALSE;
	VAT.bProbelOhneCrimpen := FALSE;
	VAT.bProbelOhneLitze := FALSE;
	
	VAT.bA55KontaktNichtGefallen := FALSE; //NBT-NEU
END_IF



//b801: BLD 130 //Sprungadresse


//L "DB6".w228_Bef_Tast_Wert DB6.DBW228 -- Befehlstasten-Wert
//L 810 //*** Magazin Leerfahren
//==I
//SPBN b810
//S "M1.3_Stop" M1.3 -- RS Stop
//StST
//S "M8.1MagLeerf" M8.1 -- Magazin Leerfahren
//R "M8.2SortLeerf" M8.2 -- Sortierer Leerfahren
//R "M8.3CrimpEinr" M8.3 -- Crimpen Einrichten
//R "M8.4NurAbisolieren" M8.4 -- Nur Abisolieren
//R "M8.5ohneKontakt" M8.5 -- Probelauf ohne Kontakt
//R "M8.6ohneCrmpen" M8.6 -- Probelauf ohne Crimpen
//R "M8.7ohneLitze" M8.7 -- Probelauf ohne Litze

//...springe nicht -> wenn gleich
IF DB6.w228_Bef_Tast_Wert = 810 THEN //*** Magazin Leerfahren
	VAT.bRsStop := TRUE; //RS Stop
	
	VAT.bMagazinLeerfahren := TRUE;
	VAT.bSortiererLeerfahren := FALSE;
	VAT.bCrimpEinrichten := FALSE;
	VAT.bNurAbisolieren := FALSE;
	VAT.bProbelOhneKontakt := FALSE;
	VAT.bProbelOhneCrimpen := FALSE;
	VAT.bProbelOhneLitze := FALSE;
END_IF

//b810: BLD 130 //Sprungadresse

//L "DB6".w228_Bef_Tast_Wert DB6.DBW228 -- Befehlstasten-Wert
//L 820 //*** Sortierer Leerfahren
//==I
//SPBN b820
//R "M1.3_Stop" M1.3 -- RS Stop

//R "M8.1MagLeerf" M8.1 -- Magazin Leerfahren
//S "M8.2SortLeerf" M8.2 -- Sortierer Leerfahren
//R "M8.3CrimpEinr" M8.3 -- Crimpen Einrichten
//R "M8.4NurAbisolieren" M8.4 -- Nur Abisolieren
//R "M8.5ohneKontakt" M8.5 -- Probelauf ohne Kontakt
//R "M8.6ohneCrmpen" M8.6 -- Probelauf ohne Crimpen
//R "M8.7ohneLitze" M8.7 -- Probelauf ohne Litze


//...springe nicht -> wenn gleich
IF DB6.w228_Bef_Tast_Wert = 820 THEN  //*** Sortierer Leerfahren
	VAT.bRsStop := FALSE; //RS Stop
	VAT.bMagazinLeerfahren := FALSE;
	VAT.bSortiererLeerfahren := TRUE;
	VAT.bCrimpEinrichten := FALSE;
	VAT.bNurAbisolieren := FALSE;
	VAT.bProbelOhneKontakt := FALSE;
	VAT.bProbelOhneCrimpen := FALSE;
	VAT.bProbelOhneLitze := FALSE;
END_IF

//b820: BLD 130 //Sprungadresse


//L "DB6".w228_Bef_Tast_Wert DB6.DBW228 -- Befehlstasten-Wert
//L 830 //*** Crimpen Einrichten
//==I
//SPBN b830
//R "M0.6" M0.6 -- SR Start
//R "M8.1MagLeerf" M8.1 -- Magazin Leerfahren
//R "M8.2SortLeerf" M8.2 -- Sortierer Leerfahren
//S "M8.3CrimpEinr" M8.3 -- Crimpen Einrichten
//R "M8.4NurAbisolieren" M8.4 -- Nur Abisolieren
//R "M8.5ohneKontakt" M8.5 -- Probelauf ohne Kontakt
//R "M8.6ohneCrmpen" M8.6 -- Probelauf ohne Crimpen
//R "M8.7ohneLitze" M8.7 -- Probelauf ohne Litze


//...springe nicht -> wenn gleich
IF DB6.w228_Bef_Tast_Wert = 830 THEN //*** Crimpen Einrichten
	VAT.bSrStart := FALSE; //SR Start
	VAT.bMagazinLeerfahren := FALSE;
	VAT.bSortiererLeerfahren := FALSE;
	VAT.bCrimpEinrichten := TRUE;
	VAT.bNurAbisolieren := FALSE;
	VAT.bProbelOhneKontakt := FALSE;
	VAT.bProbelOhneCrimpen := FALSE;
	VAT.bProbelOhneLitze := FALSE;
END_IF

//b830: BLD 130 //Sprungadresse

//L "DB6".w228_Bef_Tast_Wert DB6.DBW228 -- Befehlstasten-Wert
//L 840 //*** Nur Abisolieren
//==I
//SPBN b840
//R "M0.6" M0.6 -- SR Start
//R "M8.1MagLeerf" M8.1 -- Magazin Leerfahren
//R "M8.2SortLeerf" M8.2 -- Sortierer Leerfahren
//R "M8.3CrimpEinr" M8.3 -- Crimpen Einrichten
//S "M8.4NurAbisolieren" M8.4 -- Nur Abisolieren
//R "M8.5ohneKontakt" M8.5 -- Probelauf ohne Kontakt
//R "M8.6ohneCrmpen" M8.6 -- Probelauf ohne Crimpen
//R "M8.7ohneLitze" M8.7 -- Probelauf ohne Litze


//...springe nicht -> wenn gleich
IF DB6.w228_Bef_Tast_Wert = 840 THEN //*** Nur Abisolieren
	VAT.bSrStart := FALSE; //SR Start
	VAT.bMagazinLeerfahren := FALSE;
	VAT.bSortiererLeerfahren := FALSE;
	VAT.bCrimpEinrichten := FALSE;
	VAT.bNurAbisolieren := TRUE;
	VAT.bProbelOhneKontakt := FALSE;
	VAT.bProbelOhneCrimpen := FALSE;
	VAT.bProbelOhneLitze := FALSE;
END_IF

// b840: BLD 130 //Sprungadresse

//L "DB6".w228_Bef_Tast_Wert DB6.DBW228 -- Befehlstasten-Wert
//L 850 //*** Probelauf ohne Kontakt
//==I
//SPBN b850
//R "M0.6" M0.6 -- SR Start
//R "M8.1MagLeerf" M8.1 -- Magazin Leerfahren
//R "M8.2SortLeerf" M8.2 -- Sortierer Leerfahren
//R "M8.3CrimpEinr" M8.3 -- Crimpen Einrichten

//R "M8.4NurAbisolieren" M8.4 -- Nur Abisolieren
//S "M8.5ohneKontakt" M8.5 -- Probelauf ohne Kontakt
//R "M8.6ohneCrmpen" M8.6 -- Probelauf ohne Crimpen
//R "M8.7ohneLitze" M8.7 -- Probelauf ohne Litze


//...springe nicht -> wenn gleich
IF DB6.w228_Bef_Tast_Wert = 850 THEN  //*** Probelauf ohne Kontakt
	VAT.bSrStart := FALSE; //SR Start
	VAT.bMagazinLeerfahren := FALSE;
	VAT.bSortiererLeerfahren := FALSE;
	VAT.bCrimpEinrichten := FALSE;
	VAT.bNurAbisolieren := FALSE;
	VAT.bProbelOhneKontakt := TRUE;
	VAT.bProbelOhneCrimpen := FALSE;
	VAT.bProbelOhneLitze := FALSE;
END_IF


//b850: BLD 130 //Sprungadresse

//L "DB6".w228_Bef_Tast_Wert DB6.DBW228 -- Befehlstasten-Wert
//L 860 //*** Probelauf ohne Crimpen
//==I
//SPBN b860
//R "M0.6" M0.6 -- SR Start
//R "M8.1MagLeerf" M8.1 -- Magazin Leerfahren
//R "M8.2SortLeerf" M8.2 -- Sortierer Leerfahren
//R "M8.3CrimpEinr" M8.3 -- Crimpen Einrichten
//R "M8.4NurAbisolieren" M8.4 -- Nur Abisolieren
//R "M8.5ohneKontakt" M8.5 -- Probelauf ohne Kontakt
//S "M8.6ohneCrmpen" M8.6 -- Probelauf ohne Crimpen
//R "M8.7ohneLitze" M8.7 -- Probelauf ohne Litze


//...springe nicht -> wenn gleich
IF DB6.w228_Bef_Tast_Wert = 860 THEN //*** Probelauf ohne Crimpen
	VAT.bSrStart := FALSE; //SR Start
	VAT.bMagazinLeerfahren := FALSE;
	VAT.bSortiererLeerfahren := FALSE;
	VAT.bCrimpEinrichten := FALSE;
	VAT.bNurAbisolieren := FALSE;
	VAT.bProbelOhneKontakt := FALSE;
	VAT.bProbelOhneCrimpen := TRUE;
	VAT.bProbelOhneLitze := FALSE;
END_IF


//b860: BLD 130 //Sprungadresse

//L "DB6".w228_Bef_Tast_Wert DB6.DBW228 -- Befehlstasten-Wert
//L 870 //*** Probelauf ohne Litze
//==I
//SPBN b870
//R "M0.6" M0.6 -- SR Start
//R "M8.1MagLeerf" M8.1 -- Magazin Leerfahren
//R "M8.2SortLeerf" M8.2 -- Sortierer Leerfahren
//R "M8.3CrimpEinr" M8.3 -- Crimpen Einrichten
//R "M8.4NurAbisolieren" M8.4 -- Nur Abisolieren
//R "M8.5ohneKontakt" M8.5 -- Probelauf ohne Kontakt
//R "M8.6ohneCrmpen" M8.6 -- Probelauf ohne Crimpen
//S "M8.7ohneLitze" M8.7 -- Probelauf ohne Litze

//...springe nicht -> wenn gleich
IF DB6.w228_Bef_Tast_Wert = 870 THEN  //*** Probelauf ohne Litze
	VAT.bSrStart := FALSE; //SR Start
	VAT.bMagazinLeerfahren := FALSE;
	VAT.bSortiererLeerfahren := FALSE;
	VAT.bCrimpEinrichten := FALSE;
	VAT.bNurAbisolieren := FALSE;
	VAT.bProbelOhneKontakt := FALSE;
	VAT.bProbelOhneCrimpen := FALSE;
	VAT.bProbelOhneLitze := TRUE;
END_IF



//b870: BLD 130 //Sprungadresse
//****************************************************************************
//L 0 -- Lade die Zahl in AKKU 1 und schiebe aktuelles in AKKU 2
//T "DB6".w228_Bef_Tast_Wert DB6.DBW228 -- Befehlstasten-Wert  //Transferieren
DB6.w228_Bef_Tast_Wert := 0;

//Aend: BLD 130 //Sprungadresse
//;

END_FUNCTION

// ---- POUs/MainPous/FC3_FehlerAllg/F_ResetEndSchalterFehler.TcPOU
FUNCTION F_ResetEndSchalterFehler : BOOL
VAR_INPUT
END_VAR
VAR
END_VAR

GVL.errs.DrahthltNichtOffen := FALSE;
GVL.errs.DrahthltNichtZu := FALSE;
GVL.errs.AbisolierNichtOffen := FALSE;
GVL.errs.AbisolierNichtZu := FALSE;
GVL.errs.AbisolierNichtVorn := FALSE;
GVL.errs.AbisolierNichtRueck := FALSE;
GVL.errs.AbisolierNichtLinks := FALSE;
GVL.errs.AbisolierNichtRechts := FALSE;
GVL.errs.CrimpZangeNichtZu := FALSE;
GVL.errs.CrimpZangeNichtOffen := FALSE;
GVL.errs.CrimpeinheitNichtVorn := FALSE;
GVL.errs.CrimpeinheitNichtRueck := FALSE;
GVL.errs.KontaktSchiebenNichtVorn := FALSE;
GVL.errs.KontaktSchiebenNichtRueck := FALSE;
GVL.errs.AusstossenNichtVorn := FALSE;
GVL.errs.AusstossenNichtRueck := FALSE;

GVL.errs.DoppelMlgAbisoVornRueck := FALSE;
GVL.errs.DoppelMlgCrimpzZuOffen := FALSE;
GVL.errs.DoppelMlgCrimpEinhVornZurueck := FALSE;

END_FUNCTION

// ---- POUs/MainPous/FC4_TpKommunikation/P_TpKommunikation.TcPOU
PROGRAM P_TpKommunikation
VAR
	
END_VAR

//Netzwerk 1:
//F_AuswertungBefehlstastenVonTP(); nur noch in den Tasten-Events

//Netzwerk 2:
F_AnzeigeNiedriegePrio();

//Netzwerk 3:
//F_SignaldauerVonTastleuchte_MaschEinAuswerten();

//Netzwerk 4:
F_SAFETY_AnzeigenHohePrio_Neu();

END_PROGRAM

// ---- POUs/MainPous/FC4_TpKommunikation/F_AnzeigeNiedriegePrio.TcPOU
FUNCTION F_AnzeigeNiedriegePrio : BOOL
VAR_INPUT
END_VAR
VAR
	
	vke : BOOL;
END_VAR

//im Original, Netzwerk 2:

//U "M0.7" M0.7 -- Störung aufgetreten (gesammelt)
//SPB knp -- Springe wenn VKE = 1
IF VAT.bSammelStoerung THEN
	RETURN; //knp -- Ende der Funktion
END_IF
(*
U "T 14" T14 -- Verzög. Betriebs-Anzeigen-Reset
ON "T 3" T3 -- Fehler-Kontr.Maschine (keine Bewegung), ON: ODER NICHT
SPBN res -- Springe wenn VKE = 0

L 0
T "MW 14" MW14 -- enthäLT Betriebs-Anzeige-Bits
*)
//SPBN - Springe wenn VKE = 0 - 'jump' on FALSE equals 'do it' on TRUE
IF GVL.tonBetrAnzeigReset.Q OR NOT GVL.tonFehlerKontrMaschine.Q THEN
	GVL.BetrAnzeigeTmp := 0; //war MW14
END_IF

//res:
//L "MW 14" MW14 -- enthält Betriebs-Anzeige-Bits
//L 0 -- Aktuellen Wert als Ganzzahl in AKKU1 laden
//<>I -- 	AKKU2 ungleich AKKU1
//UN "T 14" T14 -- Verz. Betriebs-Anzeigen-Reset

vke := GVL.BetrAnzeigeTmp <> 0; //war MW14
vke := vke AND NOT GVL.tonBetrAnzeigReset.Q;

//L S5T#2S
//SE "T 14" T14 -- Verz. Betriebs-Anzeigen-Reset (SE Laden einer Zeit mit der Funktion Einschaltverzögerung),
//Zeit mit Einschaltverzögerung starten
GVL.tonBetrAnzeigReset(IN := vke, PT := T#2S);

(*
TTI@schulz-heise.com 2020-10-22:...das Ganze ist wie eine Schrittkette aufgebaut. Vor jedem der Sprünge wird der AKKU 1 geladen aber – so sieht es aus – 
nur ein Wert wird bis zum ende des Bausteins behalten, der mit dem Befehl T  DB6.DBW 226 – transferiere in das Datenwort226 des Datenbausteins 6. 
Das Programm funktioniert nur in einer STEP 7 Umgebung, da Siemens sogenannte VKE begrenzende Befehle definiert hat.
In einer anderen Umgebung müsste nach den UND Befehlen  eine Zuweisung bestehen.
*)



// Es wird eine Zahl 'mitgeschleppt', die anzeigt, wo er das letzte Mal gewesen ist...

//L 10 
GVL.BetrAnzeigeTmp := 10; // Maschine bereit, Weiter mit Taste START

//U "M0.2" M0.2 -- 2te Ablauf-Freigabe -- Aktuellen Wert als Ganzzahl in AKKU1 laden
//SPBN a16 -- Springe wenn VKE = 0

//SPBN: -> Springe wenn VKE = 0 - 'jump' on FALSE equals 'do it' on TRUE
IF VAT.bZweitAblaufFreig THEN
	//L 16
	GVL.BetrAnzeigeTmp := 16;
END_IF  

//a16: BLD 130 -- BLD sind Nulloperationen, beeinflußt die Statusbits nicht.

//U "M0.2" M0.2 -- 2te Ablauf-Freigabe
//U "M 22.7" M22.7 -- Endstellung
//SPBN a11
//L 11 //Maschine bereit zum Crimpen - Litze einführen

//SPBN: -> Springe wenn VKE = 0 - 'jump' on FALSE equals 'do it' on TRUE
IF VAT.bZweitAblaufFreig AND VAT.bEndstellung THEN
	GVL.BetrAnzeigeTmp := 11; //Maschine bereit zum Crimpen - Litze einführen
END_IF

//a11: BLD 130
//U "M0.2" M0.2 -- 2te Ablauf-Freigabe
//U "M 22.7" M22.7 -- Endstellung
//U "M11.1_Bridge_E1.1" M11.1 -- Brücke E1.1 Auslöseschalter
//SPBN a15
//L 15 //bereit zum Crimpen - Litze einführen-dann Start drücken

IF VAT.bZweitAblaufFreig AND VAT.bEndstellung AND GVL.insecAusloeseSchalter THEN
	GVL.BetrAnzeigeTmp := 15; //bereit zum Crimpen - Litze einführen-dann Start drücken
END_IF


//a15: BLD 130
//U "M0_3_Tipp" M0.3 -- Einzel-Schritt
//SPBN a6
//L 6 //Einzel-Schritt, Litze einführen

IF VAT.bEinzelSchritt THEN
	GVL.BetrAnzeigeTmp := 6; //Einzel-Schritt, Litze einführen
END_IF


//a6: BLD 130
//U "M0_3_Tipp" M0.3 -- Einzel-Schritt
//UN "M 22.7" M22.7 -- Endstellung
//SPBN a7
//L 7 //Einzel-Schritt weiter mit Start

IF VAT.bEinzelSchritt AND NOT VAT.bEndstellung THEN
	GVL.BetrAnzeigeTmp := 7; //Einzel-Schritt weiter mit Start
END_IF

//a7: BLD 130
//U "M8.3CrimpEinr" M8.3 -- Crimpen Einrichten
//SPBN a23
//L 23

IF VAT.bCrimpEinrichten THEN
	GVL.BetrAnzeigeTmp := 23; //Crimpen Einrichten
END_IF

//a23: BLD 130
//U "M 22.2" M22.2 -- 2---Vereinzelung takten od.Crimpen zu/auf Leerf-o-Ce
//UN "M 22.6" M22.6 -- Crimpen zu, bei Einstellen Leerf-o-Ce
//SPBN a13
//L 13

IF VAT.bVereinzelungTakten AND NOT VAT.bCrimpenZuBeiEinstellen THEN
	GVL.BetrAnzeigeTmp := 13;
END_IF


//a13: BLD 130
//U "M 22.2" M22.2 -- 2---Vereinzelung takten od.Crimpen zu/auf Leerf-o-Ce
//U "M 22.6" M22.6 -- Crimpen zu bei Einstellen
//Leerf-o-Ce
//SPBN a14
//L 14

IF VAT.bVereinzelungTakten AND VAT.bCrimpenZuBeiEinstellen THEN
	GVL.BetrAnzeigeTmp := 14;
END_IF

//a14: BLD 130
//U "M8.1MagLeerf" M8.1 -- Magazin Leerfahren
//SPBN a21
//L 21

IF VAT.bMagazinLeerfahren THEN
	GVL.BetrAnzeigeTmp := 21;
END_IF

//a21: BLD 130
//U "M8.2SortLeerf" M8.2 -- Sortierer Leerfahren
//SPBN a22
//L 22

IF VAT.bSortiererLeerfahren THEN
	GVL.BetrAnzeigeTmp := 22;
END_IF

//a22: BLD 130
//U "M8.4NurAbisolieren" M8.4 -- Nur Abisolieren
//SPBN a24
//L 24 //Abisolieren einrichten - Litze einführen

IF VAT.bNurAbisolieren THEN
	GVL.BetrAnzeigeTmp := 24; //Abisolieren einrichten - Litze einführen

	//U "M0.6" M0.6 -- SR Start
	//SPB a24
	//L 20 //Abisolieren einrichten - weiter mit Start
	
	IF NOT VAT.bSrStart THEN
		GVL.BetrAnzeigeTmp := 20; //Abisolieren einrichten - weiter mit Start
	END_IF

END_IF

//a24: BLD 130
//U "M8.5ohneKontakt" M8.5 -- Probelauf ohne Kontakt
//SPBN a25
//L 25

IF VAT.bProbelOhneKontakt THEN
	GVL.BetrAnzeigeTmp := 25; //Probelauf ohne Kontakt
END_IF

//a25: BLD 130
//U "M8.6ohneCrmpen" M8.6 -- Probelauf ohne Crimpen
//SPBN a26
//L 26

IF VAT.bProbelOhneCrimpen THEN
	GVL.BetrAnzeigeTmp := 26;
END_IF

//a26: BLD 130
//U "M8.7ohneLitze" M8.7 -- Probelauf ohne Litze
//SPBN a27
//L 27

IF VAT.bProbelOhneLitze THEN
	GVL.BetrAnzeigeTmp := 27;
END_IF

//a27: BLD 130
//U "M 14.0" M14.0 -- A55 Kontakt nicht gefallen
//SPBN a55
//L 55

IF VAT.bA55KontaktNichtGefallen THEN
	GVL.BetrAnzeigeTmp := 55;
END_IF

//a55: BLD 130
//T "DB6".w226_Betr_Anz_Wert DB6.DBW226 -- Betriebs-Anzeige-Wert
DB6.w226_Betr_Anz_Wert := GVL.BetrAnzeigeTmp;




//knp: BLD 130

END_FUNCTION

// ---- POUs/MainPous/FC4_TpKommunikation/F_SAFETY_AnzeigenHohePrio_Neu.TcPOU
FUNCTION F_SAFETY_AnzeigenHohePrio_Neu : BOOL (* Ehemals F_PNOZ_AnzeigenHohePrio() *)
VAR_INPUT
END_VAR
VAR
END_VAR


GVL.tonResetNotHalt(IN := NOT IO.inResetNotHalt, PT := T#2S);
IF GVL.tonResetNotHalt.Q THEN
	DB6.w226_Betr_Anz_Wert := 105; //Kein Signal von Taste Maschine-Aus
END_IF

IF GVL.tonSAFETYok.Q THEN //(ehem. T72)
	RETURN;
END_IF

DB6.w226_Betr_Anz_Wert := 127; //warte auf SAFETY-Signal...

IF NOT IO.safeOutHauptLuft THEN
		DB6.w226_Betr_Anz_Wert := 101; //Druckluft nicht ein (weiter mit Masch-Ein)
	IF NOT IO.safeOutSchutzTueren THEN
		DB6.w226_Betr_Anz_Wert := 102; //Schutztür nicht zu
	ELSIF NOT IO.safeOutNotHalt THEN
		DB6.w226_Betr_Anz_Wert := 108; //Not-Aus Steuerpult nicht OK   
	END_IF
END_IF

END_FUNCTION

// ---- POUs/MainPous/FC2_Betriebsarten/P_Betriebsarten.TcPOU
PROGRAM P_Betriebsarten
VAR
	
END_VAR

(* Baustein: FC2 - Start,Stop,Betriebsarten *)
(* FC2 - AWL2ST: Fertig *)

F_EndschalterBruecken(); // OK 

P_FlankenErzeugen(); // OK 

P_BlinktaktTastleuchten(); // OK

F_StartStopTipp(); // OK

END_PROGRAM

// ---- POUs/MainPous/FC2_Betriebsarten/F_EndschalterBruecken.TcPOU
PROGRAM F_EndschalterBruecken
VAR
	
END_VAR

(* Baustein: FC2 Start, Stop, Betriebsarten *)
(* Netzwerk: 1 Endschalter brücken *)

(* Vorgehensweise: Eine bestimmte mögliche (Ausgangs-)Kombi wird meist etwas verzögert als Eingang 'dargeboten'... 
damit wird der entsprechende Eingang simuliert *)


(*
	U "M11.0_Bridge_E1.0" M11.0 -- Brücke E1.0 Drahthalter offen
	SPBN br10
	
	UN "A 1.7" A1.7 -- Y-10 Drahthalter+Führung zu
	L S5T#500MS
	SE "Bridge_E1.0" T110 -- Brücke E1.0 Drahthalter offen
	U "Bridge_E1.0" T110 -- Brücke E1.0 Drahthalter offen
	= "E1_0" E1.0 -- R Drahthalter offen
*)
IF RVL.sBrDrahthalterIstOffen THEN //Brücke E1.2 (neu) Drahthalter offen, VAT.M11.0
	GVL.tonDrahthaltOffen(IN := NOT IO.outY10DrahthaltFuehrungZU, PT := T#500MS);
	GVL.insecDrahthalterIstOffen := GVL.tonDrahthaltOffen.Q;
ELSE

	{IF defined (CRIMP_IO_TEST)}
		GVL.insecDrahthalterIstOffen := GVL.inTmpDrahthalterIstOffen;
	{ELSE}
		GVL.insecDrahthalterIstOffen := IO.inDrahthalterIstOffen;
	{END_IF}	
	
END_IF

(*	
br10:
	U "M11.1_Bridge_E1.1" M11.1 -- Brücke E1.1 Auslöseschalter
	SPBN br11
	U "A 0.0" A0.0 -- Tastleuchte Start
	O "M0_3_Tipp" M0.3 -- Einzel-Schritt
	U "M 80.0" M80.0 -- +F E0.0 Taste Start
	= "E1_1" E1.1 -- N Auslöseschalter
*)
IF RVL.sBrAusloeseSchalter THEN //Brücke E1.3 (neu) Auslöseschalter, war VAT.M11.1
	GVL.insecAusloeseSchalter := IO.outMldTasteStart OR VAT.bEinzelSchritt AND VAT.bFlkTasteStart;
ELSE
	{IF defined (CRIMP_IO_TEST)}
		GVL.insecAusloeseSchalter := GVL.inTmpAusloeseSchalter;
	{ELSE}
		GVL.insecAusloeseSchalter := IO.inAusloeseSchalter;
	{END_IF}
END_IF
(*
br11:
	U "M11.2_Bridge_E1.2" M11.2 -- Brücke E1.2 Abisolierer zu
	SPBN br12
	U "A 1.3" A1.3 -- Y-6 Abisolierer zu
	L S5T#300MS
	SE "Bridge_E1.2" T112 -- Brücke E1.2 Abisolierer zu
	U "Bridge_E1.2" T112 -- Brücke E1.2 Abisolierer zu
	= "E1_2" E1.2 -- N Abisolierer zu
*)
IF RVL.sBrAbisoliererIstZU THEN //Brücke E1.4 (neu) Auslöseschalter, war VAT.M11.2
	GVL.tonAbisoliererIstZU(IN := IO.outY6AbisoliererZU, PT := T#300MS); // war T112
	GVL.insecAbisoliererIstZU := GVL.tonAbisoliererIstZU.Q;
ELSE	
	{IF defined (CRIMP_IO_TEST)}
		GVL.insecAbisoliererIstZU := GVL.inTmpAbisoliererIstZU;
	{ELSE}
		GVL.insecAbisoliererIstZU := IO.inAbisoliererIstZU;
	{END_IF}
END_IF
(*
br12: U "M11.3_Bridge_E1.3" M11.3 -- Brücke E1.3 Abisolierer vorn
	SPBN br13
	UN "A 1.5" A1.5 -- Y-8 Abisolierer rück
	L S5T#300MS
	SE "Bridge_E1.3" T113 -- Brücke E1.3 Abisolierer vorn
	U "Bridge_E1.3" T113 -- Brücke E1.3 Abisolierer vorn
	= "E1_3" E1.3 -- R Abisolierer vorn
*)
IF RVL.sBrAbisoliererIstVORN THEN //Brücke E1.5 (neu) Abisolierer vorn, war VAT.M11.3
	GVL.tonAbisoliererIstVORN(IN := NOT IO.outY8AbisoliererRUECK, PT := T#300MS); // war T113
	GVL.insecAbisoliererIstVORN := GVL.tonAbisoliererIstVORN.Q;
ELSE
	{IF defined (CRIMP_IO_TEST)}
		GVL.insecAbisoliererIstVORN := GVL.inTmpAbisoliererIstVORN;
	{ELSE}	
		GVL.insecAbisoliererIstVORN := IO.inAbisoliererIstVORN;
	{END_IF}	
END_IF
(*
br13: U "M11.4_Bridge_E1.4" M11.4 -- Brücke E1.4 Abisolierer rück (abisoliert)
	SPBN br14
	U "A 1.5" A1.5 -- Y-8 Abisolierer rück
	L S5T#400MS
	SE "Bridge_E1.4" T114 -- Brücke E1.4 Abisolierer rück (abisoliert)
	U "Bridge_E1.4" T114 -- Brücke E1.4 Abisolierer rück (abisoliert)
	= "E1_4" E1.4 -- R Abisolierer rück (abisoliert)
*)
IF RVL.sBrAbisoliererIstRUECK THEN //Brücke E1.6 (neu) Abisolierer rück (abisoliert), war VAT.M11.4
	GVL.tonAbisoliererIstRUECK(IN := IO.outY8AbisoliererRUECK, PT := T#400MS); // war T114
	GVL.insecAbisoliererIstRUECK := GVL.tonAbisoliererIstRUECK.Q;
ELSE
	{IF defined (CRIMP_IO_TEST)}
		GVL.insecAbisoliererIstRUECK := GVL.inTmpAbisoliererIstRUECK;
	{ELSE}	
		GVL.insecAbisoliererIstRUECK := IO.inAbisoliererIstRUECK;
	{END_IF}	
END_IF
(*
br14: U "M11.5_Bridge_E1.5" M11.5 -- Brücke E1.5 Abisolierer links (aus Arbeitsraum)
	SPBN br15
	U "A 1.2" A1.2 -- Y-5 Abisolierer nach links+Abdeckung zu
	L S5T#500MS
	SE "Bridge_E1.5" T115 -- Brücke E1.5 Abisolierer links (aus Arbeitsraum)
	U "Bridge_E1.5" T115 -- Brücke E1.5 Abisolierer links (aus Arbeitsraum)
	= "E1_5" E1.5 -- R Abisolierer links (aus Arbeitsraum)
*)
IF RVL.sBrAbisoliererIstLINKS THEN //Brücke E1.7 (neu) Abisolierer links (aus Arbeitsraum), war VAT.M11.5
	GVL.tonAbisoliererIstLINKS(IN := IO.outY5AbisolierNachLINKS, PT := T#500MS); // war T115
	GVL.insecAbisoliererIstLINKS := GVL.tonAbisoliererIstLINKS.Q;
ELSE
	{IF defined (CRIMP_IO_TEST)}
		GVL.insecAbisoliererIstLINKS := GVL.inTmpAbisoliererIstLINKS;
	{ELSE}	
		GVL.insecAbisoliererIstLINKS := IO.inAbisoliererIstLINKS;
	{END_IF}	
END_IF
(*
br15: U "M11.6_Bridge_E1.6" M11.6 -- Brücke E1.6 Crimpzange zu
	SPBN br16
	U "A 1.6" A1.6 -- Y-9 Crimpen zu
	L S5T#600MS
	SE "Bridge_E1.6" T116 -- Brücke E1.6 Crimpzange zu
	U "Bridge_E1.6" T116 -- Brücke E1.6 Crimpzange zu
	= "E1_6" E1.6 -- N Crimpzange zu
*)
IF RVL.sBrCrimpZangeIstZU THEN //Brücke E1.8 (neu) Crimpzange zu, war VAT.M11.6
	GVL.tonCrimpZangeIstZU(IN := IO.outY9CrimperZU, PT := T#600MS); // war T116
	GVL.insecCrimpZangeIstZU := GVL.tonCrimpZangeIstZU.Q;
ELSE	
	{IF defined (CRIMP_IO_TEST)}
		GVL.insecCrimpZangeIstZU := GVL.inTmpCrimpZangeIstZU;
	{ELSE}	
		GVL.insecCrimpZangeIstZU := IO.inCrimpZangeIstZU;
	{END_IF}
END_IF
(*
br16: U "M11.7_Bridge_E1.7" M11.7 -- Brücke E1.7 Crimpzange offen
	SPBN br17
	UN "A 1.6" A1.6 -- Y-9 Crimpen zu
	L S5T#400MS
	SE "Bridge_E1.7" T117 -- Brücke E1.7 Crimpzange offen
	U "Bridge_E1.7" T117 -- Brücke E1.7 Crimpzange offen
	= "E1_7" E1.7 -- R Crimpzange offen
*)
IF RVL.sBrCrimpZangeIstOFFEN THEN //Brücke E1.9 (neu) Crimpzange offen, war VAT.M11.7
	GVL.tonCrimpZangeIstOFFEN(IN := NOT IO.outY9CrimperZU, PT := T#400MS); // war T117
	GVL.insecCrimpZangeIstOFFEN := GVL.tonCrimpZangeIstOFFEN.Q;
ELSE
	{IF defined (CRIMP_IO_TEST)}
		GVL.insecCrimpZangeIstOFFEN := GVL.inTmpCrimpZangeIstOFFEN;
	{ELSE}	
		GVL.insecCrimpZangeIstOFFEN := IO.inCrimpZangeIstOFFEN;
	{END_IF}	
END_IF
(*
br17: U "M12.0_Bridge_E2.0" M12.0 -- Brücke E2.0 Kontakt gefallen
	SPBN br20
	U "M 21.7" M21.7 -- Kontakt-Anforderung
	L S5T#500MS
	SE "Bridge_E2.0" T120 -- Brücke E2.0 Kontakt gefallen
	U "Bridge_E2.0" T120 -- Brücke E2.0 Kontakt gefallen
	= "E2_0" E2.0 -- L Kontakt gefallen
*)
IF RVL.sBrKontaktIstGefallen THEN //Brücke E1.10 (neu) Kontakt gefallen, war VAT.M12.0
	GVL.tonBrKontaktIstGefallen(IN := VAT.bKontaktAnforderung, PT := T#500MS); // war T120 -> M21.7
	GVL.insecKontaktIstGefallen := GVL.tonBrKontaktIstGefallen.Q;
ELSE	
	{IF defined (CRIMP_IO_TEST)}
		GVL.insecKontaktIstGefallen := GVL.inTmpKontaktIstGefallen;
	{ELSE}	
		GVL.insecKontaktIstGefallen := IO.inKontaktIstGefallen;
	{END_IF}
END_IF
(*
br20: U "M12.1_Bridge_E2.1" M12.1 -- Brücke E2.1 Crimpeinheit vorn
	SPBN br21
	U "A 1.1" A1.1 -- Y-4 Crimpeinheit vor
	L S5T#300MS
	SE "Bridge_E2.1" T121 -- Brücke E2.1 Crimpeinheit vorn
	U "Bridge_E2.1" T121 -- Brücke E2.1 Crimpeinheit vorn
	= "E2_1" E2.1 -- R Crimpeinheit vorn
*)
IF RVL.sBrCrimpEinheitIstVORN THEN //Brücke E1.11 (neu) Crimpeinheit vorn, war VAT.M12.1
	GVL.tonCrimpEinheitIstVORN(IN := IO.outY4CrimpEinheitVOR, PT := T#300MS); // war T121
	GVL.insecCrimpEinheitIstVORN := GVL.tonCrimpEinheitIstVORN.Q;
ELSE	
	{IF defined (CRIMP_IO_TEST)}
		GVL.insecCrimpEinheitIstVORN := GVL.inTmpCrimpEinheitIstVORN;
	{ELSE}	
		GVL.insecCrimpEinheitIstVORN := IO.inCrimpEinheitIstVORN;
	{END_IF}	
END_IF
(*
br21: U "M12.2_Bridge_E2.2" M12.2 -- Brücke E2.2 Kontakt-Schieben vorn
	SPBN br22
	U "A 1.0" A1.0 -- Y-3 Kontakt-Schieben
	L S5T#400MS
	SE "Bridge_E2.2" T122 -- Brücke E2.2 Kontakt-Schieben vorn
	U "Bridge_E2.2" T122 -- Brücke E2.2 Kontakt-Schieben vorn
	= "E2_2" E2.2 -- R Kontakt-Schieben vorn
*)
IF RVL.sBrKontaktSchiebenVORN THEN //Brücke E1.14 (neu) Kontakt-Schieben vorn, war VAT.M12.2
	GVL.tonKontaktSchiebenVORN(IN := IO.outY3KontaktSchieben, PT := T#400MS); // war T122
	GVL.insecKontaktSchiebenVORN := GVL.tonKontaktSchiebenVORN.Q;
ELSE	
	{IF defined (CRIMP_IO_TEST)}
		GVL.insecKontaktSchiebenVORN := GVL.inTmpKontaktSchiebenVORN;
	{ELSE}
		GVL.insecKontaktSchiebenVORN := IO.inKontaktSchiebenVORN;
	{END_IF}
END_IF
(*
br22: U "M12.3_Bridge_E2.3" M12.3 -- Brücke E2.3 Ausstoßen vorn
	SPBN br23
	U "A 0.6" A0.6 -- Y-1 Ausstoßen
	L S5T#300MS
	SE "Bridge_E2.3" T123 -- Brücke E2.3 Ausstoßen vorn
	U "Bridge_E2.3" T123 -- Brücke E2.3 Ausstoßen vorn
	= "E2_3" E2.3 -- R Ausstoßen vorn
*)
IF RVL.sBrAusstossenVORN THEN //Brücke E1.13 (neu) Ausstoßen vorn, war VAT.M12.3
	GVL.tonAusstossenVORN(IN := IO.outY1Ausstossen, PT := T#300MS); // war T123
	GVL.insecAusstossenVORN := GVL.tonAusstossenVORN.Q;
ELSE
	{IF defined (CRIMP_IO_TEST)}
		GVL.insecAusstossenVORN := GVL.inTmpAusstossenVORN;
	{ELSE}	
		GVL.insecAusstossenVORN := IO.inAusstossenVORN;
	{END_IF}
END_IF
(*
br23: U "M12.4_Bridge_E2.4" M12.4 -- Brücke E2.4 Crimpeinheit rück
	SPBN br24
	UN "A 1.1" A1.1 -- Y-4 Crimpeinheit vor
	L S5T#400MS
	SE "Bridge_E2.4" T124 -- Brücke E2.4 Crimpeinheit rück
	U "Bridge_E2.4" T124 -- Brücke E2.4 Crimpeinheit rück
	= "E2_4" E2.4 -- R Crimpeinheit rück
*)
IF RVL.sBrAusstossenVORN THEN //Brücke E1.12 (neu) Crimpeinheit rück, war VAT.M12.4
	GVL.tonCrimpEinheitIstRUECK(IN := IO.outY4CrimpEinheitVOR, PT := T#300MS); // war T124
	GVL.insecCrimpEinheitIstRUECK := GVL.tonCrimpEinheitIstRUECK.Q;
ELSE
	{IF defined (CRIMP_IO_TEST)}
		GVL.insecCrimpEinheitIstRUECK := GVL.inTmpCrimpEinheitIstRUECK;
	{ELSE}
		GVL.insecCrimpEinheitIstRUECK := IO.inCrimpEinheitIstRUECK;
	{END_IF}	
END_IF
(*
br24: U "M12.5_Bridge_E2.5" M12.5 -- Brücke E2.5 Magazin gefüllt
	SPBN br25
	U "E2_5" E2.5 -- N Magazin gefüllt
	= "E2_5" E2.5 -- N Magazin gefüllt
*)
IF RVL.sBrMagazinGEFUELLT THEN // //Brücke E1.15 (neu) Magazin gefüllt, war VAT.M12.5
	GVl.insecMagazinGEFUELLT := IO.inMagazinGEFUELLT; //???
ELSE	
	{IF defined (CRIMP_IO_TEST)}
		GVL.insecMagazinGEFUELLT := GVL.inTmpMagazinGEFUELLT;
	{ELSE}
		GVl.insecMagazinGEFUELLT := IO.inMagazinGEFUELLT;
	{END_IF}	
END_IF
(*
br25: BLD 130
*)

END_PROGRAM

// ---- POUs/MainPous/FC2_Betriebsarten/P_FlankenErzeugen.TcPOU
PROGRAM P_FlankenErzeugen
VAR
	akk1, akk2 : DWORD;
	dwTmp : DWORD;
END_VAR

(* Netzwerk: 2 Flanken erzeugen *)


//...wird offensichtlich nicht verwendet!	
(*
L "DB6".d0 DB6.DBD0 -- Zuw.v. -- altes Eingangsdoppelwort aus DB6-RAM nach AKKU1
INVD -- 1-Komplement Ganzzahl (32 Bit)
*)
//akk1 := NOT DB6.d0;
(*
L ED 0  -- L ED 0 schiebe AKKU1 nach AKKU2 und Lade Eingangsdoppelwort 0 in AKKU1
T "DB6".d0 DB6.DBD0 -- Zuw.v. -- rette aktuelles Eingangsdoppelwort in DB6-RAM
*)
//akk2 := akk1;
//akk1 := dwTmp; //Das müsste das original Eingangsdoppelwort 0 sein.
//DB6.d0 := akk1;
(*
UD -- UND-Doppelwort Akku1 mit Akku 2, Das Ergebnis wird in AKKU 1 gespeichert.
T "MD 80" MD80 -- +Fs ED0 -- das Statuswort wird nicht beeinflusst
*) 
//GVL.MD80 := (akk1 AND akk2); //+Fs ED0


//ToDo, Frage: ----------------- Wirkt jetzt Akku1 noch nach? ------------------
//sehr wahrscheinlich nicht.
//ansonsten ist das alles unnötig...
(*
UN "M8.1MagLeerf" M8.1 -- Magazin Leerfahren
UN "M8.2SortLeerf" M8.2 -- Sortierer Leerfahren
UN "M8.3CrimpEinr" M8.3 -- Crimpen Einrichten
UN "M8.4NurAbisolieren" M8.4 -- Nur Abisolieren
UN "M8.5ohneKontakt" M8.5 -- Probelauf ohne Kontakt
UN "M8.6ohneCrmpen" M8.6 -- Probelauf ohne Crimpen
UN "M8.7ohneLitze" M8.7 -- Probelauf ohne Litze
= "M8.0NormalCrimp" M8.0 -- Normal Crimpen
*)

VAT.bNormalCrimp :=	NOT VAT.bMagazinLeerfahren AND //Magazin Leerfahren
				NOT VAT.bSortiererLeerfahren AND //Sortierer Leerfahren
				NOT VAT.bCrimpEinrichten AND //Crimpen Einrichten
				NOT VAT.bNurAbisolieren AND //Nur Abisolieren
				NOT VAT.bProbelOhneKontakt AND //Probelauf ohne Kontakt
				NOT VAT.bProbelOhneCrimpen AND //Probelauf ohne Crimpen
				NOT VAT.bProbelOhneLitze; 	  //Probelauf ohne Litze

END_PROGRAM

// ---- POUs/MainPous/FC2_Betriebsarten/P_BlinktaktTastleuchten.TcPOU
PROGRAM P_BlinktaktTastleuchten
VAR
	//locByte0 : BYTE;
	blink:FB_MY_BLINK;
	blinkOld:BOOL := FALSE;
	b1HzOld:BOOL;
END_VAR

(* Netzwerk: 3 Blinktakt Tastleuchten - OK *)

//125 ms sind 8 Hz, mal sehen, ob ich die überhaupt brauche
blink(bEn := TRUE, udiTiOn_ms := 62, udiTiOff_ms := 63);

VAT.b1HzFlanke := FALSE;

IF blink.bQ <> blinkOld THEN
		
	VAT.byBlinkTakt := VAT.byBlinkTakt + 1;
	
	IO.outMldTasteStart :=	VAT.byBlinkTakt.0 AND // 8-Hz Blinktakt
							VAT.byBlinkTakt.1 AND // 4-Hz Blinktakt
							VAT.byBlinkTakt.2 AND // 2-Hz Blinktakt
							VAT.bEinzelSchritt
						 OR
							VAT.bSrStart AND
							NOT VAT.bSammelStoerung;
	
							
							
							
	IF b1HzOld <> VAT.byBlinkTakt.3 THEN
		VAT.b1HzFlanke := VAT.byBlinkTakt.3; //todo noch keine flanke
	END_IF	
	b1HzOld := VAT.byBlinkTakt.3;

	IF DB6.diStueck_Vorwahl > DB6.diStueck_Fertig THEN
		DB6.diStueck_Noch := DB6.diStueck_Vorwahl - DB6.diStueck_Fertig;
	END_IF						
END_IF

blinkOld := blink.bQ;

//IO.outResA1_2 := VAT.b1HzFlanke;


IF NOT VAT.b1HzFlanke THEN
	RETURN;
END_IF

//Verl. 5 Minuten für Betriebstunden-Zähler, todo Warum?

 


(*
	
		(*
			L 0
			T "MB 5" MB5 -- +F Blinktakt-Generator
		*)	
		VAT.M5 := 0;	
		(*	
			U "T 0" T0 -- Taktgeber
			SPB Takt -- Springe wenn VKE = 1
		*)	
		IF NOT GVL.T0.Q THEN
			(*
				L S5T#60MS
				SA "T 0" T0 -- Taktgeber
				CLR
				SA "T 0" T0 -- Taktgeber
			*)
			GVL.T0(IN := TRUE, PT := T#60MS);
			(*	
				L "MB 4" MB4 -- Blinktakt-Generator
				T LB 0
				INC 1
				T "MB 4" MB4 -- Blinktakt-Generator
				
				L LB 0
				INVI
				L "MB 4" MB4 -- Blinktakt-Generator
				UW
				
				T "MB 5" MB5 -- +F Blinktakt-Generator
			*)
			locByte0 := VAT.M4;
			VAT.M4 := VAT.M4 + 1;
			locByte0 := NOT locByte0;
			VAT.M5 := locByte0 AND VAT.M4;
			
			(*	
				U "M 4.0" M4.0 -- 8-Hz Blinktakt
				U "M 4.1" M4.1 -- 4-Hz Blinktakt
				U "M 4.2" M4.2 -- 2-Hz Blinktakt
				U "M0_3_Tipp" M0.3 -- Einzel-Schritt
				O "M0.6" M0.6 -- SR Start
				UN "M0.7" M0.7 -- Störung aufgetreten (gesammelt)
				= "A 0.0" A0.0 -- Tastleuchte Start
			*)	
			IO.outMldTasteStart :=	VAT.M4.0 AND // 8-Hz Blinktakt
									VAT.M4.1 AND // 4-Hz Blinktakt
									VAT.M4.2 AND // 2-Hz Blinktakt
									VAT.M0.3 OR  // Einzel-Schritt   
									VAT.M0.6 AND // SR Start
									NOT VAT.M0.7; // Störung aufgetreten (gesammelt)
			(*	
				L "DB6".d64Stueck_Vorwahl DB6.DBD64 -- Stückzahl-Vorwahl Stückz
				L "DB6".d68Stueck_Fertig DB6.DBD68 -- Fertig Stückz
				<D -- AKKU2 kleiner als AKKU1
				SPB Takt
				
				-D -- AKKU1 von AKKU2 subtrahieren
				T "DB6".d72Stueck_Noch DB6.DBD72 -- Noch Stückzahl
			*)
			IF DB6.d64Stueck_Vorwahl > DB6.d68Stueck_Fertig THEN
				DB6.d72Stueck_Noch := DB6.d64Stueck_Vorwahl - DB6.d68Stueck_Fertig;
			END_IF
		ELSE
			GVL.T0(IN := FALSE);	
		END_IF	//end if NOT GVL.T0.Q...
		
		(*	
		Takt: BLD 130
			U "M 5.3" M5.3 -- +F 1-Hz Blinktakt
			SPBN bz
		*)	
		IF NOT VAT.M5.3 THEN
			RETURN;
		END_IF
*)


		
(*
	U "T 34" T34 -- Verl. 5 Minuten für Betriebstunden-Zähler
	SPBN bz
*)
IF NOT GVL.tofBetrStdZaehl.Q THEN
	RETURN;
END_IF
	
(*	
	L "DB6".d160 DB6.DBD160 -- Betriebs-Sekunden
	+ L#1
	T "DB6".d160 DB6.DBD160 -- Betriebs-Sekunden
	L L#3600
	<D -- AKKU2 kleiner als AKKU1
	SPB bz
*)
	
DB6.runTime.seconds := DB6.runTime.seconds + 1;
IF DB6.runTime.seconds < 3600 THEN
	RETURN;
END_IF
	
(*	
	L 0
	T "DB6".d160 DB6.DBD160 -- Betriebs-Sekunden
*)	
DB6.runTime.seconds := 0;
(*	
	L "DB6".d164_Betriebs_St DB6.DBD164 -- Betriebs-Stunden
	+ L#1
	T "DB6".d164_Betriebs_St DB6.DBD164 -- Betriebs-Stunden
*)
DB6.runTime.hours := DB6.runTime.hours  + 1;
(*	
bz: BLD 130
*)

END_PROGRAM

// ---- POUs/Helper/FB_MY_BLINK.TcPOU
FUNCTION_BLOCK FB_MY_BLINK
VAR_INPUT
	bEn : BOOL;
	udiTiOn_ms : UDINT := 100;
	udiTiOff_ms : UDINT := 100;
END_VAR
VAR_OUTPUT
	bQ : BOOL;
END_VAR
VAR
	state : WORD := 0;
	enTiOn : BOOL := FALSE;
	TiOn : TON;
	enTiOff : BOOL := FALSE;
	TiOff : TON;
END_VAR

CASE state OF
	0:
		IF bEn THEN
			state := 1;
			enTiOn := TRUE;
			bQ := TRUE;
		END_IF
	1:
		IF TiOn.Q THEN
			bQ := FALSE;
			enTiOn := FALSE;
			IF bEn THEN
				state := 2;
				enTiOff := TRUE;
			ELSE	
				state := 0;		
				enTiOff := FALSE;
			END_IF
		END_IF
	2:
		IF TiOff.Q THEN
			enTiOff := FALSE;
			IF bEn THEN
				state := 1;
				enTiOn := TRUE;
				bQ := TRUE;
			ELSE
				state := 0;
				enTiOn := FALSE;
				bQ := FALSE;
			END_IF
		END_IF
END_CASE
	
TiOn(IN := enTiOn, PT := UDINT_TO_TIME(udiTiOn_ms));

TiOff(IN := enTiOff, PT := UDINT_TO_TIME(udiTiOff_ms));

END_FUNCTION_BLOCK

// ---- POUs/MainPous/FC2_Betriebsarten/F_StartStopTipp.TcPOU
FUNCTION F_StartStopTipp : BOOL
VAR_INPUT
END_VAR
VAR
	bTmp:BOOL;
END_VAR

(* Netzwerk: 4 Start, Stop, Tipp... *)

(*
U "T 19" T19 -- Kontaktauswurf nach Einschalten
U "M8.4NurAbisolieren" M8.4 -- Nur Abisolieren
O "M 80.0" M80.0 -- +F E0.0 Taste Start
S "M0.6" M0.6 -- SR Start -- /ER geht auf 0 !!!
R "M1.3_Stop" M1.3 -- RS Stop StST -- /ER geht auf 0 !!!
UN "M0.7" M0.7 -- Störung aufgetreten (gesammelt)
= "M0.5" M0.5 -- Bedingung für Ablauf-Freigabe
*)

//VAT.bFlkTasteStart set in P_InputHandling() -- NBT-NEU
	
IF (GVL.tsvKontauswurf.Q AND VAT.bNurAbisolieren) OR VAT.bFlkTasteStart THEN	
	VAT.bSrStart := TRUE;
	VAT.bRsStop := FALSE;
END_IF

VAT.bAblaufFreigabe := NOT VAT.bSammelStoerung;

(*
O "M0_3_Tipp" M0.3 -- Einzel-Schritt
ON "M0.5" M0.5 -- Bedingung für Ablauf-Freigabe
O "M1.3_Stop" M1.3 -- RS Stop
R "M0.6" M0.6 -- SR Start -- R (Rücksetze Bit) schreibt bei VKE = 1 (und MCR = 1) den Wert "0" in das adressierte Bit.
							-- Bei MCR = 0 wird das adressierte Bit nicht verändert.
*)
			
IF VAT.bEinzelSchritt OR NOT VAT.bAblaufFreigabe OR VAT.bRsStop THEN	
	VAT.bSrStart := FALSE;
END_IF

(*							-- /ER geht auf 0 !!!
U "M0.6" M0.6 -- SR Start
O "M 80.0" M80.0 -- +F E0.0 Taste Start
U "M0.5" M0.5 -- Bedingung für Ablauf-Freigabe
= "M0.2" M0.2 -- 2te Ablauf-Freigabe
*)


VAT.bZweitAblaufFreig := (VAT.bSrStart OR VAT.bFlkTasteStart) AND VAT.bAblaufFreigabe;

END_FUNCTION

// ---- POUs/MainPous/F20_Ablauf/P_Ablauf.TcPOU
PROGRAM P_Ablauf
VAR
	ErrNo : WORD;
	endstellungOk : BOOL;
	fbAllesInSollpos : FB_AllesInSollposition;
	AblaufketteNormal : FB_AblaufketteNormal;
END_VAR

(*
FC20 Ablauf
Zeitstempel Code: 11.01.2019 13:17:50
Interface: 16.02.2009 10:58:19
*)

fbAllesInSollpos(errorOffset := 500); //OK
GVL.SolPosErrorIdx := fbAllesInSollpos.nErrNo;

//Nur wenn SafetyFALSE UND Taste Start > 1 Sek.
P_AblaufReset(); //OK - mit Abweichung / auskomm.

AblaufketteNormal(); //OK

F_AblaufketteLeerfahren(); //OK

endstellungOk := F_Endstellung();

F_Ventile(); //OK

END_PROGRAM

// ---- POUs/MainPous/F20_Ablauf/FB_AllesInSollposition.TcPOU
FUNCTION_BLOCK FB_AllesInSollposition
VAR_INPUT
	errorOffset : WORD := 0;
END_VAR
	
VAR_OUTPUT
	bError : BOOL;
	nErrNo : WORD;
	bErrMute : BOOL;
END_VAR

VAR
	fehlerBlocker : TSV;
END_VAR

(* Netzwerk: 1 Alles in Sollposition *)
nErrNo := 0;
bError := TRUE;
(*

UN "A 0.6" A0.6 -- Y-1 Ausstoßen
UN "E2_3" E2.3 -- R Ausstoßen vorn
O
U "A 0.6" A0.6 -- Y-1 Ausstoßen
U "E2_3" E2.3 -- R Ausstoßen vorn
= "M 3.0" M3.0 -- Alles in Sollposition
*)
//VAT0.M3.0 := (NOT IO.a06Ausstossen AND NOT IO.e23AusstossenVorn) OR
//			(IO.a06Ausstossen AND IO.e23AusstossenVorn);

VAT.bAllesInSollPos	:=	(NOT IO.outY1Ausstossen AND NOT GVL.insecAusstossenVORN) OR
						(IO.outY1Ausstossen AND GVL.insecAusstossenVORN);	
			
			
			
(*
UN "A 1.0" A1.0 -- Y-3 Kontakt-Schieben
U "E2_2" E2.2 -- R Kontakt-Schieben vorn
R "M 3.0" M3.0 -- (Rücksetzen, wenn VKE 1 ist) Alles in Sollposition
*)
//IF NOT IO.a10KontaktSchieben AND IO.e22KontaktSchiebenVorn THEN
//	VAT0.M3.0 := FALSE;
//END_IF
IF NOT IO.outY3KontaktSchieben AND GVL.insecKontaktSchiebenVORN THEN
	VAT.bAllesInSollPos := FALSE;
	nErrNo := errorOffset + 1;
	M_BlockTimer();
	RETURN;
END_IF

(*
U "A 1.0" A1.0 -- Y-3 Kontakt-Schieben
UN "E2_2" E2.2 -- R Kontakt-Schieben vorn
R "M 3.0" M3.0 -- Alles in Sollposition
*)
//IF IO.a10KontaktSchieben AND NOT IO.e22KontaktSchiebenVorn THEN
//	VAT0.M3.0 := FALSE;
//END_IF
IF IO.outY3KontaktSchieben AND NOT GVL.insecKontaktSchiebenVORN THEN
	VAT.bAllesInSollPos := FALSE;
	nErrNo := errorOffset + 2;
	M_BlockTimer();
	RETURN;
END_IF
(*
O "E2_1" E2.1 -- R Crimpeinheit vorn
ON "E2_4" E2.4 -- R Crimpeinheit rück
UN "A 1.1" A1.1 -- Y-4 Crimpeinheit vor
R "M 3.0" M3.0 -- Alles in Sollposition
*)
//IF IO.e21CrimpEinheitVorn OR NOT IO.e24CrimpeinheitRueck AND NOT IO.a11CrimpeinheitVor THEN
//	VAT0.M3.0 := FALSE;
//END_IF
IF (GVL.insecCrimpEinheitIstVORN OR NOT GVL.insecCrimpEinheitIstRUECK) AND NOT IO.outY4CrimpEinheitVOR THEN
	VAT.bAllesInSollPos := FALSE;
	nErrNo := errorOffset + 3;
	M_BlockTimer();
	RETURN;
END_IF

(*
ON "E2_1" E2.1 -- R Crimpeinheit vorn
O "E2_4" E2.4 -- R Crimpeinheit rück
U "A 1.1" A1.1 -- Y-4 Crimpeinheit vor
R "M 3.0" M3.0 -- Alles in Sollposition
*)
//IF NOT GVL.e21CrimpEinheitVorn OR IO.e24CrimpeinheitRueck AND IO.a11CrimpeinheitVor THEN
//	VAT0.M3.0 := FALSE;
//END_IF
IF (NOT GVL.insecCrimpEinheitIstVORN OR GVL.insecCrimpEinheitIstRUECK) AND IO.outY4CrimpEinheitVOR THEN
	VAT.bAllesInSollPos := FALSE;
	nErrNo := errorOffset + 4;
	M_BlockTimer();
	RETURN;
END_IF
(*
U "E1_5" E1.5 -- R Abisolierer links (aus Arbeitsraum)
UN "A 1.2" A1.2 -- Y-5 Abisolierer nach links+Abdeckung zu
R "M 3.0" M3.0 -- Alles in Sollposition
*)
//IF IO.e15AbisoliererLinks AND NOT IO.a12AbisoliererNachLi THEN
//	VAT0.M3.0 := FALSE;
//END_IF
IF GVL.insecAbisoliererIstLINKS AND NOT IO.outY5AbisolierNachLINKS THEN
	VAT.bAllesInSollPos := FALSE;
	nErrNo := errorOffset + 5;
	M_BlockTimer();
	RETURN;
END_IF
(*
UN "E1_5" E1.5 -- R Abisolierer links (aus Arbeitsraum)
U "A 1.2" A1.2 -- Y-5 Abisolierer nach links+Abdeckung zu
R "M 3.0" M3.0 -- Alles in Sollposition
*)
//IF NOT IO.e15AbisoliererLinks AND IO.a12AbisoliererNachLi THEN
//VAT0.M3.0 := FALSE;
//END_IF
IF NOT GVL.insecAbisoliererIstLINKS AND IO.outY5AbisolierNachLINKS THEN
	VAT.bAllesInSollPos := FALSE;
	nErrNo := errorOffset + 6;
	M_BlockTimer();
	RETURN;
END_IF
(*
U "E1_2" E1.2 -- N Abisolierer zu
UN "A 1.3" A1.3 -- Y-6 Abisolierer zu
R "M 3.0" M3.0 -- Alles in Sollposition
*)
//IF IO.e12AbisoliererZu AND NOT IO.a13AbisoliererZu THEN
//	VAT0.M3.0 := FALSE;
//END_IF
IF GVL.insecAbisoliererIstZU AND NOT IO.outY6AbisoliererZU THEN
	VAT.bAllesInSollPos := FALSE;
	nErrNo := errorOffset + 7;
	M_BlockTimer();
	RETURN;
END_IF
(*
UN "E1_2" E1.2 -- N Abisolierer zu
U "A 1.3" A1.3 -- Y-6 Abisolierer zu
R "M 3.0" M3.0 -- Alles in Sollposition
*)
//IF NOT IO.e12AbisoliererZu AND IO.a13AbisoliererZu THEN
//	VAT0.M3.0 := FALSE;
//END_IF
IF NOT GVL.insecAbisoliererIstZU AND IO.outY6AbisoliererZU THEN
	VAT.bAllesInSollPos := FALSE;
	nErrNo := errorOffset + 8;
	M_BlockTimer();
	RETURN;
END_IF
(*
ON "E1_3" E1.3 -- R Abisolierer vorn
O "E1_4" E1.4 -- R Abisolierer rück (abisoliert)
UN "A 1.5" A1.5 -- Y-8 Abisolierer rück
R "M 3.0" M3.0 -- Alles in Sollposition
*)

IF (NOT GVL.insecAbisoliererIstVORN OR GVL.insecAbisoliererIstRUECK) AND NOT IO.outY8AbisoliererRUECK THEN
	VAT.bAllesInSollPos := FALSE;
	nErrNo := errorOffset + 9;
	M_BlockTimer();
	RETURN;
END_IF
(*
O "E1_3" E1.3 -- R Abisolierer vorn
ON "E1_4" E1.4 -- R Abisolierer rück (abisoliert)
U "A 1.5" A1.5 -- Y-8 Abisolierer rück
R "M 3.0" M3.0 -- Alles in Sollposition
*)

IF (GVL.insecAbisoliererIstVORN OR NOT GVL.insecAbisoliererIstRUECK) AND IO.outY8AbisoliererRUECK THEN
	VAT.bAllesInSollPos := FALSE;
	nErrNo := errorOffset + 10;
	M_BlockTimer();
	RETURN;
END_IF
(*
// O E 1.6
ON "E1_7" E1.7 -- R Crimpzange offen
UN "A 1.6" A1.6 -- Y-9 Crimpen zu
R "M 3.0" M3.0 -- Alles in Sollposition
*)
//IF NOT IO.e17CrimpzangeOffen AND NOT IO.a16CrimpenZu THEN
//	VAT0.M3.0 := FALSE;
//END_IF
IF NOT GVL.insecCrimpZangeIstOFFEN AND NOT IO.outY9CrimperZU THEN
	VAT.bAllesInSollPos := FALSE;
	nErrNo := errorOffset + 11;
	M_BlockTimer();
	RETURN;
END_IF
(*
ON "E1_6" E1.6 -- N Crimpzange zu
O "E1_7" E1.7 -- R Crimpzange offen
U "A 1.6" A1.6 -- Y-9 Crimpen zu
R "M 3.0" M3.0 -- Alles in Sollposition
*)
//IF NOT IO.e16CrimpzangeZu OR IO.e17CrimpzangeOffen AND IO.a16CrimpenZu THEN
//	VAT0.M3.0 := FALSE;
//END_IF
IF (NOT GVL.insecCrimpZangeIstZU OR GVL.insecCrimpZangeIstOFFEN) AND IO.outY9CrimperZU THEN
	VAT.bAllesInSollPos := FALSE;
	nErrNo := errorOffset + 12;
	M_BlockTimer();
	RETURN;
END_IF
(*
UN "E1_0" E1.0 -- R Drahthalter offen
UN "A 1.7" A1.7 -- Y-10 Drahthalter+Führung zu
R "M 3.0" M3.0 -- Alles in Sollposition
*)
//IF NOT IO.e10DrahthalterOffen AND NOT IO.a17DrahthalterUndFuehrungZu THEN
//	VAT0.M3.0 := FALSE;
//END_IF
IF NOT GVL.insecDrahthalterIstOffen AND NOT IO.outY10DrahthaltFuehrungZU THEN
	VAT.bAllesInSollPos := FALSE;
	nErrNo := errorOffset + 13;
	M_BlockTimer();
	RETURN;
END_IF
(*
U "E1_0" E1.0 -- R Drahthalter offen
U "A 1.7" A1.7 -- Y-10 Drahthalter+Führung zu
R "M 3.0" M3.0 -- Alles in Sollposition
*)
//IF IO.e10DrahthalterOffen AND IO.a17DrahthalterUndFuehrungZu THEN
//	VAT0.M3.0 := FALSE;
//END_IF
IF GVL.insecDrahthalterIstOffen AND IO.outY10DrahthaltFuehrungZU THEN
	VAT.bAllesInSollPos := FALSE;
	nErrNo := errorOffset + 14;
	M_BlockTimer();
	RETURN;
END_IF

fehlerBlocker(IN := FALSE);
bErrMute := fehlerBlocker.Q;
bError := FALSE;

METHOD PRIVATE M_BlockTimer : BOOL
VAR_INPUT
END_VAR
fehlerBlocker(IN := TRUE, PT := T#800MS);
bErrMute := fehlerBlocker.Q;
END_METHOD

END_FUNCTION_BLOCK

// ---- POUs/Helper/TSV.TcPOU
FUNCTION_BLOCK TSV

VAR_INPUT
	IN : BOOL;
	PT : TIME := T#2s;
END_VAR
VAR_OUTPUT
	Q : BOOL;
END_VAR
VAR
	rTrig : R_TRIG;
	tonTime : TON;
	
END_VAR

(*
SV-Verhalten [AWL-SV gibt es in ST nicht, deshalb dieser Nachbau]:
SV <Zeit> startet die adressierte Zeit, wenn das VKE von "0" auf "1" wechselt. Die programmierte
Zeitdauer läuft ab, auch wenn das VKE inzwischen auf "0" wechselt. Wechselt das VKE von "0" auf
"1", bevor die programmierte Zeit abgelaufen ist, wird die programmierte Zeitdauer neu gestartet.
*)

rTrig(CLK := IN);
IF rTrig.Q THEN
	tonTime(IN := FALSE, PT := PT);
	Q := TRUE;
END_IF

tonTime(IN := Q, PT := PT);

IF tonTime.Q THEN
	Q := FALSE;
END_IF

END_FUNCTION_BLOCK

// ---- POUs/MainPous/F20_Ablauf/FB_AblaufketteNormal.TcPOU
FUNCTION_BLOCK FB_AblaufketteNormal
VAR_INPUT
END_VAR
VAR_OUTPUT
END_VAR
VAR
	dwTest:DWORD;
	dwTest2:DWORD;
	nTmp:INT;
	
	rtgAusloeseSchalt : R_TRIG;
	rtgEinzelschritt : R_TRIG;
	einzelSchrittOffset : WORD := 400;
END_VAR


rtgAusloeseSchalt(CLK := GVL.insecAusloeseSchalter);
VAT.bFlankeAusloeseschalter := rtgAusloeseSchalt.Q;


rtgEinzelschritt(CLK := VAT.bEinzelSchritt);
IF rtgEinzelschritt.Q THEN
	GVL.EinzelschrittIdx := einzelSchrittOffset + 20; //NBT-NEU: Einzelschritt - Start
END_IF


//Timer muss immer durchlaufen werden. TOF kann permanent auf FALSE gelassen werden, wenn er eine Start-Flanke erhalten hat.
GVL.tofAblVerzProbelauf(IN := FALSE);


//Timer hier hin verlegt von:
//*** 8---Ausstoßen vor
//Grund: Timer muss immer durchlaufen werden.
//DB6.nAusstossverz := 1500; //Test später raus.
GVL.tonAusstoss(IN := VAT.bCrZangeAUF_AisolierVOR, PT := INT_TO_TIME (DB6.nAusstossverz)); 


//Timer muss immer durchlaufen werden. TOF kann permanent auf FALSE gelassen werden, wenn er eine Start-Flanke erhalten hat.
GVL.tofBetrStdZaehl(IN := FALSE);


(* Netzwerk: 3 Ablaufkette normal *)

	(*
		U "M 22.7" M22.7 -- Endstellung, //Erstabfrage, Ergebnis wird ins VKE geschrieben
		SPBN s0 -- Springe wenn VKE = 0
		
		O "M 81.1" M81.1 -- +F E1.1 Auslöseschalter
		O "M8.5ohneKontakt" M8.5 -- Probelauf ohne Kontakt
		O "M8.6ohneCrmpen" M8.6 -- Probelauf ohne Crimpen
		O "M8.7ohneLitze" M8.7 -- Probelauf ohne Litze
		SPBN s0
			
		O "M0_3_Tipp" M0.3 -- Einzel-Schritt
		O "M0.2" M0.2 -- 2te Ablauf-Freigabe
		U "M 3.0" M3.0 -- Alles in Sollposition
		UN "T 20" T20 -- Ablauf-Verz.bei Probelauf
		SPBN s0
	*)

	
//SPBN -> Springe wenn VKE = 0 -> 'Springe bei FALSE' heißt 'Tu was bei TRUE'.
IF VAT.bEndstellung THEN 
	//SPBN -> Springe wenn VKE = 0 -> 'Springe bei FALSE' heißt 'Tu was bei TRUE'.
	IF VAT.bFlankeAusloeseschalter OR VAT.bProbelOhneKontakt OR VAT.bProbelOhneCrimpen OR VAT.bProbelOhneLitze THEN  
		//SPBN -> Springe wenn VKE = 0 -> 'Springe bei FALSE' heißt 'Tu was bei TRUE'.
		//VAT.bZweitAblaufFreig := (VAT.bSrStart OR VAT.bFlkTasteStart) AND VAT.bAblaufFreigabe in F_StartStopTipp()...
		IF (VAT.bEinzelSchritt OR VAT.bZweitAblaufFreig) AND VAT.bAllesInSollPos AND NOT GVL.tofAblVerzProbelauf.Q THEN
			MAIN.M_Log(reqLevel:=CVL.TRACE, objectName:= 'Ablauf', sMsg:= 'START',errNo := 16#FFFFFFFF);			
			(*
			S "M 20.0" M20.0 -- 0---Drahthalter + Drahtführung zu, Setze M20.0 auf 1, wenn VKE 1 ist
			*)
			VAT.bDrahtHalterUndFuehrungZU := TRUE; //Start der Kette Abisolierer zu
			GVL.EinzelschrittIdx := einzelSchrittOffset + 21; //NBT-NEU: Drahthalter + Drahtführung zu
			(*	
			UN "M8.4NurAbisolieren" M8.4 -- Nur Abisolieren
			UN "M8.5ohneKontakt" M8.5 -- Probelauf ohne Kontakt
			S "M 21.7" M21.7 -- Kontakt-Anforderung, Setze M21.7 auf 1, wenn VKE 1 ist, setze Erstabfragebit /ER zurück
			*)
			IF NOT VAT.bNurAbisolieren AND NOT VAT.bProbelOhneKontakt THEN
				MAIN.M_Log(reqLevel:=CVL.TRACE, objectName:= 'SET', sMsg:= 'bKontaktAnforderung',errNo := 16#FFFFFFFF);
				VAT.bKontaktAnforderung := TRUE;
			END_IF
			(*
			U "M8.6ohneCrmpen" M8.6 -- Probelauf ohne Crimpen -- Erstabfrage, Ergebnis wird ins VKE geschrieben
			= "M 21.6" M21.6 -- Aktueller Ablauf ohne Crimpen, -- = <Bit> schreibt (bei MCR = 1) das VKE in das adressierte Bit
			SPA end -- Absoluter Sprung zur Sprungmarke 'end'
			*)
			
			VAT.bAktAblaufOhneCr := VAT.bProbelOhneCrimpen;

			RETURN;

		END_IF

	END_IF

END_IF
	
(*
s0: BLD 130

	U "M0.2" M0.2 -- 2te Ablauf-Freigabe
	U "M 3.0" M3.0 -- Alles in Sollposition
	SPBN end -- springe wenn VKE = "0" nach 'end'
*)
//VAT.bZweitAblaufFreig := (VAT.bSrStart OR VAT.bFlkTasteStart) AND VAT.bAblaufFreigabe in F_StartStopTipp()...	
IF (VAT.bZweitAblaufFreig AND VAT.bAllesInSollPos) = FALSE THEN
	RETURN;
END_IF
	
(*	
	//*** 1--- Abisolierer zu
	U "M 20.0" M20.0 -- 0---Drahthalter + Drahtführung zu
	R "M 20.0" M20.0 -- 0---Drahthalter + Drahtführung zu
	S "M 20.1" M20.1 -- 1---Abisolierer zu
	SPB end  -- Springe wenn VKE = 1
*)
IF VAT.bDrahtHalterUndFuehrungZU THEN
	VAT.bDrahtHalterUndFuehrungZU := FALSE;
	VAT.bAbisoliererZU := TRUE; //M20.1
	GVL.EinzelschrittIdx := einzelSchrittOffset + 22; //NBT-NEU: Abisolierer zu
	MAIN.M_Log(reqLevel:=CVL.TRACE, objectName:= 'Ablauf', sMsg:= '1--- Abisolierer zu',errNo := 16#FFFFFFFF);
	RETURN;
END_IF


(*	
	//*** 2---Abisolierer rück (abisolieren)
	U "M 20.1" M20.1 -- 1---Abisolierer zu, Erstabfrage, Ergebnis wird ins VKE geschrieben
	R "M 20.1" M20.1 -- 1---Abisolierer zu, wenn VKE 1 ist
	S "M 20.2" M20.2 -- 2---Abisolierer rück (abisolieren), wenn VKE 1 ist
	// SA <Zeit> startet die adressierte Zeit, wenn das VKE von "1" auf "0" wechselt. 
	L S5T#5M
	SA "T 34" T34 -- Verl. 5 Minuten für Betriebstunden-Zähler, Laden einer Zeit mit der Funktion Ausschaltverzögerung
	SPB end  -- Springe wenn VKE = 1
*)	
	IF VAT.bAbisoliererZU THEN
		VAT.bAbisoliererZU := FALSE; //M20.1
		VAT.bAbisoliererRUECK := TRUE; //M20.2
		//Zeit mit Ausschaltverzögerung starten
		GVL.tofBetrStdZaehl(IN := VAT.bAbisoliererRUECK, PT := T#5M);
		GVL.EinzelschrittIdx := einzelSchrittOffset + 23; //NBT-NEU: Abisolierer rück (abisolieren)
		MAIN.M_Log(reqLevel:=CVL.TRACE, objectName:= 'Ablauf', sMsg:= '2---Abisolierer rück',errNo := 16#FFFFFFFF);
		RETURN;
	END_IF
	//GVL.tofBetrStdZaehl(IN := VAT.bAbisoliererRUECK, PT := T#5M); //Timer muss durchlaufen werden! Checken
	
(*	
	//*** 3---Abisolierer nach links + Abisolierer auf
	U "M 20.2" M20.2 -- 2---Abisolierer rück (abisolieren)
	SPBN s3  -- Springe wenn VKE = 0
*)
	IF VAT.bAbisoliererRUECK THEN //M20.2
	(*	
		U "M 21.7" M21.7 -- Kontakt-Anforderung --- Erstabfrage, Ergebnis wird ins VKE geschrieben
		S "M 14.0" M14.0 -- A55 Kontakt nicht gefallen, Setzen des Operanden M14.0, wenn VKE 1 ist, setze Erstabfragebit /ER zurück
		SPB s3 -- Springe wenn VKE = 1
		*)
		
		IF VAT.bKontaktAnforderung THEN //M21.7
			MAIN.M_Log(reqLevel:=CVL.TRACE, objectName:= 'FB_AblaufketteNormal', sMsg:= 'bKontaktAnforderung = TRUE',errNo := 16#FFFFFFFF);
			VAT.bA55KontaktNichtGefallen := TRUE; //M14.0
			// Springe wenn VKE = 1 zu s3
		ELSE
			MAIN.M_Log(reqLevel:=CVL.TRACE, objectName:= 'FB_AblaufketteNormal', sMsg:= 'bKontaktAnforderung = FALSE',errNo := 16#FFFFFFFF);	
			//ToDo: Welche Erstabfrage, VKE sollte hier eigentlich immer 0 sein...?
			//damit kein Setzen ??
			
			VAT.bA55KontaktNichtGefallen := FALSE;
			
			//S (Setze Bit) schreibt bei VKE = 1 und bei eingeschaltetem Master Control Relay (MCR = 1) den Wert
			//"1" in das adressierte Bit.
			(*
			R "M 20.2" M20.2 -- 2---Abisolierer rück (abisolieren), Rücksetzen des Operanden M20.2, wenn VKE 1 ist
			S "M 20.3" M20.3 -- 3---Abisolierer nach links + Abisolierer auf, Setzen des Operanden M20.3, wenn VKE 1 ist
			*)
			
			VAT.bAbisoliererRUECK := FALSE;
			VAT.bAbisoliererLINKSundAUF := TRUE;
			GVL.EinzelschrittIdx := einzelSchrittOffset + 24; //NBT-NEU: Abisolierer nach links + Abisolierer auf
			
			(*
			U "M8.4NurAbisolieren" M8.4 -- Nur Abisolieren --- Erstabfrage, Ergebnis wird ins VKE geschrieben
			L S5T#1S
			SA "T 20" T20 -- Zeit mit Ausschaltverzögerung starten, Ablauf-Verz. bei Probelauf, 
			

			CLR -- VKE auf 0 setzen
			SA "T 20" T20 -- Ablauf-Verz.bei Probelauf, startet die adressierte Zeit, wenn das VKE von "1" auf "0" wechselt.
			SPA end

			*)
			GVL.tofAblVerzProbelauf(IN := VAT.bNurAbisolieren, PT := T#1S); //T20
			MAIN.M_Log(reqLevel:=CVL.TRACE, objectName:= 'Ablauf', sMsg:= '3---Abisolierer links/auf',errNo := 16#FFFFFFFF);
			RETURN;
		
		END_IF
	
	END_IF

(*	
s3: BLD 130

	//*** 4---Crimpeinheit vor
	U "M 20.3" M20.3 -- 3---Abisolierer nach links + Abisolierer auf
	UN "M8.4NurAbisolieren" M8.4 -- Nur Abisolieren
	R "M 20.3" M20.3 -- 3---Abisolierer nach links + Abisolierer auf, Rücksetzen des Operanden M20.3, wenn VKE 1 ist
	S "M 20.4" M20.4 -- 4---Crimpeinheit vor, Setzen des Operanden M20.4, wenn VKE 1 ist
	SPB end
*)

